// TIA Portal V18 program export: 1 tag tables, 1 data types, 3 data blocks, 17 code blocks (in call order from the OBs), 10 instance data blocks

VAR_GLOBAL   // PLC tag table "默认变量表"
   Room1_ES1 AT %I200.0 : Bool;
   Room1_ES2 AT %I200.1 : Bool;
   Room1_ES3 AT %I200.2 : Bool;
   Room1_ES4 AT %I200.3 : Bool;
   Room1_ES5 AT %I206.0 : Bool;
   Room1Control_ES6 AT %I206.1 : Bool;
   "Room1_Key1.1" AT %I206.2 : Bool;
   "Room1Control_Key1.1" AT %I206.3 : Bool;
   "Room1_door1.1" AT %I212.0 : Bool;
   Room2_ES1 AT %I218.0 : Bool;
   Room2_ES2 AT %I218.1 : Bool;
   Room2_ES3 AT %I218.2 : Bool;
   Room2_ES4 AT %I218.3 : Bool;
   Room2_ES5 AT %I224.0 : Bool;
   Room2Control_ES6 AT %I224.1 : Bool;
   "Room2_Key1.1" AT %I224.2 : Bool;
   "Room2Control_Key1.1" AT %I224.3 : Bool;
   "Room2_door1.1" AT %I230.0 : Bool;
   ACC_ES1 AT %I236.0 : Bool;
   ACC_ES2 AT %I236.1 : Bool;
   ACC_ES3 AT %I236.2 : Bool;
   ACC_ES4 AT %I236.3 : Bool;
   "ACC_Key1.1" AT %I242.2 : Bool;
   "ACCControl_Key1.1" AT %I242.3 : Bool;
   "ACC_door1.1" AT %I248.0 : Bool;
   "ACC_door2.1" AT %I248.1 : Bool;
   VerticalBeam_ES1 AT %I254.0 : Bool;   // vertical beam ES
   VerticalBeam_ES2 AT %I254.1 : Bool;
   VerticalBeam_ES3 AT %I254.2 : Bool;
   VerticalBeam_ES4 AT %I254.3 : Bool;
   "VerticalBeam_Key1.1" AT %I260.2 : Bool;
   "VerticalBeamControl_Key1.1" AT %I260.3 : Bool;
   "VerticalBeam_door1.1" AT %I266.0 : Bool;
   "VerticalBeam_door2.1" AT %I266.1 : Bool;
   Room1_SB1 AT %I100.0 : Bool;   // 搜索清场按钮1
   Room1_SB2 AT %I100.1 : Bool;
   Room2_SB1 AT %I100.4 : Bool;
   Room2_SB2 AT %I100.5 : Bool;
   ACC_SB1 AT %I101.0 : Bool;
   ACC_SB2 AT %I101.1 : Bool;
   VerticalBeam_SB1 AT %I101.4 : Bool;
   VerticalBeam_SB2 AT %I101.5 : Bool;
   ACC_Ready AT %I102.0 : Bool;
   ACC_Run AT %I102.1 : Bool;
   ACC_StopBeam AT %I102.2 : Bool;
   ACC_Stop AT %I102.3 : Bool;
   ACC_Fault AT %I102.4 : Bool;
   ACC_Mode1 AT %I102.5 : Bool;   // 治疗室1、加速器2、垂直束
   ACC_Mode2 AT %I102.6 : Bool;   // 治疗室2、加速器2、垂直束
   ACC_Mode3 AT %I102.7 : Bool;   // 加速器2、垂直束
   EnvironmentalMonitoring1 AT %I103.4 : Bool;
   EnvironmentalMonitoring2 AT %I103.5 : Bool;
   EnvironmentalMonitoring3 AT %I103.6 : Bool;
   EnvironmentalMonitoring4 AT %I103.7 : Bool;
   Room1_AudibleAlarm AT %Q100.0 : Bool;
   Room1_StrobeLamp1 AT %Q100.1 : Bool;
   Room1_StrobeLamp2 AT %Q100.2 : Bool;
   Room1_Red AT %Q100.5 : Bool;   // 禁止进入指示灯
   Room1_Yellow AT %Q100.6 : Bool;   // 限制进入指示灯
   Room1_Green AT %Q100.7 : Bool;   // 控制进入指示灯
   Room1_Door1NoEntry AT %Q101.0 : Bool;   // 门禁1禁止进入
   Room1_Door1RestrictedEntry AT %Q101.1 : Bool;   // 门禁1限制进入
   Room1_Door1ControlEntry AT %Q101.2 : Bool;   // 门禁1控制进入
   "Room1_door1.2" AT %I212.4 : Bool;
   "Room1_Key1.2" AT %I206.6 : Bool;
   "Room1Control_Key1.2" AT %I206.7 : Bool;
   "Room2_Key1.2" AT %I224.6 : Bool;
   "Room2Control_Key1.2" AT %I224.7 : Bool;
   "Room2_door1.2" AT %I230.4 : Bool;
   "ACC_Key1.2" AT %I242.6 : Bool;
   "ACCControl_Key1.2" AT %I242.7 : Bool;
   "VerticalBeam_Key1.2" AT %I260.6 : Bool;
   "VerticalBeamControl_Key1.2" AT %I260.7 : Bool;
   "VerticalBeam_door1.2" AT %I266.4 : Bool;
   "VerticalBeam_door2.2" AT %I266.5 : Bool;
   "ACC_door1.2" AT %I248.4 : Bool;
   "ACC_door2.2" AT %I248.5 : Bool;
   ACC_Interlock1 AT %Q400.0 : Bool;
   ACC_Interlock2 AT %Q400.1 : Bool;
   RF_Interlock1 AT %Q400.2 : Bool;
   RF_Interlock2 AT %Q400.3 : Bool;
   IonSource_Interlock1 AT %Q400.4 : Bool;
   IonSource_Interlock2 AT %Q400.5 : Bool;
   MIS__Interlock1 AT %Q400.6 : Bool;
   MIS__Interlock2 AT %Q400.7 : Bool;
   Room1_ES1_ValueStatus AT %I201.0 : Bool;
   Room1_ES2_ValueStatus AT %I201.1 : Bool;
   Room1_ES3_ValueStatus AT %I201.2 : Bool;
   Room1_ES4_ValueStatus AT %I201.3 : Bool;
   Room1_ES5_ValueStatus AT %I207.0 : Bool;
   Room1Control_ES6_ValueStatus AT %I207.1 : Bool;
   "Room1_Key1.1_ValueStatus" AT %I207.2 : Bool;
   "Room1Control_Key1.1_ValueStatus" AT %I207.3 : Bool;
   "Room1_Key1.2_ValueStatus" AT %I207.6 : Bool;
   "Room1Control_Key1.2_ValueStatus" AT %I207.7 : Bool;
   "Room1_door1.1_ValueStatus" AT %I213.0 : Bool;
   "Room1_door1.2_ValueStatus" AT %I213.4 : Bool;
   Room2_ES1_ValueStatus AT %I219.0 : Bool;
   Room2_ES2_ValueStatus AT %I219.1 : Bool;
   Room2_ES3_ValueStatus AT %I219.2 : Bool;
   Room2_ES4_ValueStatus AT %I219.3 : Bool;
   Room2_ES5_ValueStatus AT %I225.0 : Bool;
   Room2Control_ES6_ValueStatus AT %I225.1 : Bool;
   "Room2_Key1.1_ValueStatus" AT %I225.2 : Bool;
   "Room2Control_Key1.1_ValueStatus" AT %I225.3 : Bool;
   "Room2_Key1.2_ValueStatus" AT %I225.6 : Bool;
   "Room2Control_Key1.2_ValueStatus" AT %I225.7 : Bool;
   "Room2_door1.1_ValueStatus" AT %I231.0 : Bool;
   "Room2_door1.2_ValueStatus" AT %I231.4 : Bool;
   ACC_ES1_ValueStatus AT %I237.0 : Bool;
   ACC_ES2_ValueStatus AT %I237.1 : Bool;
   ACC_ES3_ValueStatus AT %I237.2 : Bool;
   ACC_ES4_ValueStatus AT %I237.3 : Bool;
   "ACC_Key1.1_ValueStatus" AT %I243.2 : Bool;
   "ACCControl_Key1.1_ValueStatus" AT %I243.3 : Bool;
   "ACC_Key1.2_ValueStatus" AT %I243.6 : Bool;
   "ACCControl_Key1.2_ValueStatus" AT %I243.7 : Bool;
   "ACC_door1.1_ValueStatus" AT %I249.0 : Bool;
   "ACC_door2.1_ValueStatus" AT %I249.1 : Bool;
   "ACC_door1.2_ValueStatus" AT %I249.4 : Bool;
   "ACC_door2.2_ValueStatus" AT %I249.5 : Bool;
   VerticalBeam_ES1_ValueStatus AT %I255.0 : Bool;
   VerticalBeam_ES2_ValueStatus AT %I255.1 : Bool;
   VerticalBeam_ES3_ValueStatus AT %I255.2 : Bool;
   VerticalBeam_ES4_ValueStatus AT %I255.3 : Bool;
   "VerticalBeam_Key1.1_ValueStatus" AT %I261.2 : Bool;
   "VerticalBeamControl_Key1.1_ValueStatus" AT %I261.3 : Bool;
   "VerticalBeam_Key1.2_ValueStatus" AT %I261.6 : Bool;
   "VerticalBeamControl_Key1.2_ValueStatus" AT %I261.7 : Bool;
   "VerticalBeam_door1.1_ValueStatus" AT %I267.0 : Bool;
   "VerticalBeam_door2.1_ValueStatus" AT %I267.1 : Bool;
   "VerticalBeam_door1.2_ValueStatus" AT %I267.4 : Bool;
   "VerticalBeam_door2.2_ValueStatus" AT %I267.5 : Bool;
   ACC_Interlock1_ValueStatus AT %I400.0 : Bool;
   ACC_Interlock2_ValueStatus AT %I400.1 : Bool;
   RF_Interlock1_ValueStatus AT %I400.2 : Bool;
   RF_Interlock2_ValueStatus AT %I400.3 : Bool;
   IonSource_Interlock1_ValueStatus AT %I400.4 : Bool;
   IonSource_Interlock2_ValueStatus AT %I400.5 : Bool;
   MIS__Interlock1_ValueStatus AT %I400.6 : Bool;
   MIS__Interlock2_ValueStatus AT %I400.7 : Bool;
   Room2_AudibleAlarm AT %Q102.0 : Bool;
   Room2_StrobeLamp1 AT %Q102.1 : Bool;
   Room2_StrobeLamp2 AT %Q102.2 : Bool;
   Room2_Red AT %Q102.5 : Bool;
   Room2_Yellow AT %Q102.6 : Bool;
   Room2_Green AT %Q102.7 : Bool;
   Room2_Door1NoEntry AT %Q103.0 : Bool;
   Room2_Door1RestrictedEntry AT %Q103.1 : Bool;
   Room2_Door1ControlEntry AT %Q103.2 : Bool;
   ACC_AudibleAlarm AT %Q104.0 : Bool;
   ACC_StrobeLamp1 AT %Q104.1 : Bool;
   ACC_StrobeLamp2 AT %Q104.2 : Bool;
   ACC_Red AT %Q104.5 : Bool;
   ACC_Yellow AT %Q104.6 : Bool;
   ACC_Green AT %Q104.7 : Bool;
   ACC_StrobeLamp3 AT %Q104.3 : Bool;
   ACC_StrobeLamp4 AT %Q104.4 : Bool;
   ACC_Door1NoEntry AT %Q105.0 : Bool;
   ACC_Door1RestrictedEntry AT %Q105.1 : Bool;
   ACC_Door1ControlEntry AT %Q105.2 : Bool;
   ACC_Door2NoEntry AT %Q105.3 : Bool;
   ACC_Door2RestrictedEntry AT %Q105.4 : Bool;
   ACC_Door2ControlEntry AT %Q105.5 : Bool;
   VerticalBeam_AudibleAlarm AT %Q106.0 : Bool;
   VerticalBeam_StrobeLamp1 AT %Q106.1 : Bool;
   VerticalBeam_StrobeLamp2 AT %Q106.2 : Bool;
   VerticalBeam_StrobeLamp3 AT %Q106.3 : Bool;
   VerticalBeam_StrobeLamp4 AT %Q106.4 : Bool;
   VerticalBeam_Red AT %Q106.5 : Bool;
   VerticalBeam_Yellow AT %Q106.6 : Bool;
   VerticalBeam_Green AT %Q106.7 : Bool;
   VerticalBeam_Door1NoEntry AT %Q107.0 : Bool;
   VerticalBeam_Door1RestrictedEntry AT %Q107.1 : Bool;
   VerticalBeam_Door1ControlEntry AT %Q107.2 : Bool;
   VerticalBeam_Door2NoEntry AT %Q107.3 : Bool;
   VerticalBeam_Door2RestrictedEntry AT %Q107.4 : Bool;
   VerticalBeam_Door2ControlEntry AT %Q107.5 : Bool;
   Room1_AreaReady AT %Q108.0 : Bool;   // 治疗室1控制区就绪
   Room2_AreaReady AT %Q108.1 : Bool;   // 治疗室2控制区就绪
   ACC_AreaReady AT %Q108.2 : Bool;   // 加速器2控制区就绪
   Room1_StartAlarm AT %Q101.7 : Bool;
   Room2_StartAlarm AT %Q103.7 : Bool;
   ACC_StartAlarm AT %Q105.7 : Bool;
   VerticalBeam_StartAlarm AT %Q107.7 : Bool;
   Room1_BeamAllowed AT %Q108.4 : Bool;   // 允许治疗室1打靶
   Room2_BeamAllowed AT %Q108.5 : Bool;   // 允许治疗室2打靶
   ACC_BeamAllowed AT %Q108.6 : Bool;   // 允许加速器出束
   VerticalBeam_AreaReady AT %Q108.3 : Bool;   // 垂直束控制区就绪
END_VAR

TYPE "FIODia"
// stored: IsFailsafeCompliant true
   STRUCT
      ModulePassOut : Bool;   // 模块钝化
      ModuleACK_REQ : Bool;   // 模块需确认重新集成
      Channel0PassOut : Bool;   // 通道0钝化
      Channel1PassOut : Bool;   // 通道1钝化
      Channel2PassOut : Bool;   // 通道2钝化
      Channel3PassOut : Bool;   // 通道3钝化
      Channel4PassOut : Bool;   // 通道4钝化
      Channel5PassOut : Bool;   // 通道5钝化
      Channel6PassOut : Bool;   // 通道6钝化
      Channel7PassOut : Bool;   // 通道7钝化
   END_STRUCT;
END_TYPE

DATA_BLOCK "数据块_1"   // DB2
{ S7_Optimized_Access := 'TRUE' }
VERSION : 0.1
// stored: AutoNumber true, DBAccessibleFromOPCUA true, IsOnlyStoredInLoadMemory false, IsRetainMemResEnabled false, IsWriteProtectedInAS false, MemoryReserve 100
   VAR
      Room1_Interlock : Bool;
      Room2_Interlock : Bool;
      ACC_Interlock : Bool;
      VerticalBeam_Interlock : Bool;
      Interlock : Bool;
   END_VAR
BEGIN
END_DATA_BLOCK

DATA_BLOCK "数据块_2"   // DB3
{ S7_Optimized_Access := 'TRUE' }
VERSION : 0.1
// stored: AutoNumber true, DBAccessibleFromOPCUA true, IsOnlyStoredInLoadMemory false, IsRetainMemResEnabled false, IsWriteProtectedInAS false, MemoryReserve 100
   VAR
      "F-DI_A21_1" : "FIODia";   // 安全输入模块A21.1
      "F-DI_A21_2" { S7_SetPoint := 'True'} : "FIODia";   // 安全输入模块A21.2
      "F-DI_A21_3" { S7_SetPoint := 'True'} : "FIODia";   // 安全输入模块A21.3
      "F-DI_A21_4" { S7_SetPoint := 'True'} : "FIODia";   // 安全输入模块A21.4
      "F-DI_A21_5" { S7_SetPoint := 'True'} : "FIODia";   // 安全输入模块A21.5
      "F-DI_A21_6" { S7_SetPoint := 'True'} : "FIODia";   // 安全输入模块A21.6
      "F-DI_A21_7" { S7_SetPoint := 'True'} : "FIODia";   // 安全输入模块A21.7
      "F-DI_A21_8" { S7_SetPoint := 'True'} : "FIODia";   // 安全输入模块A21.8
      "F-DI_A21_9" { S7_SetPoint := 'True'} : "FIODia";   // 安全输入模块A21.9
      "F-DI_A21_10" { S7_SetPoint := 'True'} : "FIODia";   // 安全输入模块A21.10
      "F-DI_A21_11" { S7_SetPoint := 'True'} : "FIODia";   // 安全输入模块A21.11
      "F-DI_A21_12" { S7_SetPoint := 'True'} : "FIODia";   // 安全输入模块A21.12
      "F-DQ_A21_1" { S7_SetPoint := 'True'} : "FIODia";   // 安全输出模块A22.1
      "F-DQ_A21_2" { S7_SetPoint := 'True'} : "FIODia";   // 安全输出模块A22.2
   END_VAR
BEGIN
END_DATA_BLOCK

DATA_BLOCK "EPICSData"   // DB8
{ S7_Optimized_Access := 'FALSE'; DB_Accessible_From_OPC_UA := 'FALSE' }
VERSION : 0.1
// stored: AutoNumber true, DBAccessibleFromOPCUA false, IsOnlyStoredInLoadMemory false, IsWriteProtectedInAS false
   VAR
      Reset : Bool;
   END_VAR
BEGIN
END_DATA_BLOCK

ORGANIZATION_BLOCK "Main"   // OB1, LAD, ProgramCycle
TITLE = "Main Program Sweep (Cycle)"
{ S7_Optimized_Access := 'TRUE' }
VERSION : 0.1
// stored: AutoNumber true, IsIECCheckEnabled false, SetENOAutomatically false
   VAR_INPUT
      Initial_Call : Bool;   // Initial call of this OB
      Remanence : Bool;   // =True, if remanent data are available
   END_VAR
BEGIN

REGION Network 2
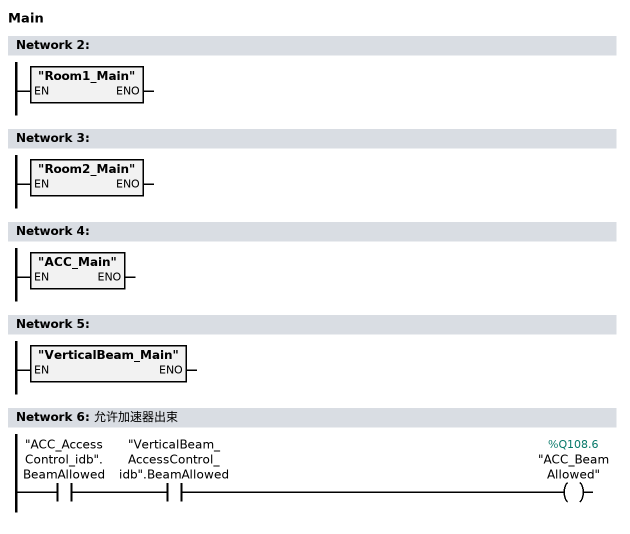
   RUNG wire#powerrail
      "Room1_Main"()
   END_RUNG
   // the same network as SCL:
   "Room1_Main"();
END_REGION

REGION Network 3
   RUNG wire#powerrail
      "Room2_Main"()
   END_RUNG
   // the same network as SCL:
   "Room2_Main"();
END_REGION

REGION Network 4
   RUNG wire#powerrail
      "ACC_Main"()
   END_RUNG
   // the same network as SCL:
   "ACC_Main"();
END_REGION

REGION Network 5
   RUNG wire#powerrail
      "VerticalBeam_Main"()
   END_RUNG
   // the same network as SCL:
   "VerticalBeam_Main"();
END_REGION

REGION Network 6: 允许加速器出束
   RUNG wire#powerrail
      Contact( "ACC_AccessControl_idb".BeamAllowed )
      Contact( "VerticalBeam_AccessControl_idb".BeamAllowed )
      Coil( "ACC_BeamAllowed" )
   END_RUNG
   // the same network as SCL:
   "ACC_BeamAllowed" := "ACC_AccessControl_idb".BeamAllowed AND "VerticalBeam_AccessControl_idb".BeamAllowed;
END_REGION
END_ORGANIZATION_BLOCK

FUNCTION "Room1_Main" : Void   // FC4, LAD
{ S7_Optimized_Access := 'TRUE' }
VERSION : 0.1
// stored: AutoNumber true, IsIECCheckEnabled false, SetENOAutomatically false, UDAEnableTagReadback false
BEGIN

REGION Network 1: 区域搜索
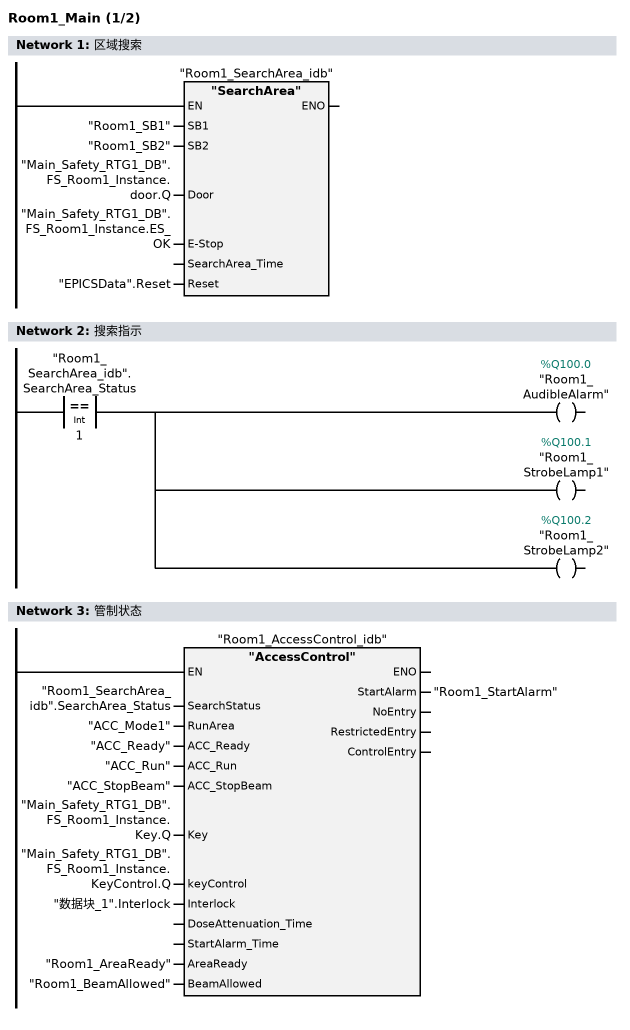
   RUNG wire#powerrail
      "Room1_SearchArea_idb"(SB1 := "Room1_SB1", SB2 := "Room1_SB2", Door := "Main_Safety_RTG1_DB".FS_Room1_Instance.door.Q, "E-Stop" := "Main_Safety_RTG1_DB".FS_Room1_Instance.ES_OK, SearchArea_Time :=, Reset := "EPICSData".Reset)
   END_RUNG
   // the same network as SCL:
   "Room1_SearchArea_idb"(SB1 := "Room1_SB1",   // "SearchArea"
                          SB2 := "Room1_SB2",
                          Door := "Main_Safety_RTG1_DB".FS_Room1_Instance.door.Q,
                          "E-Stop" := "Main_Safety_RTG1_DB".FS_Room1_Instance.ES_OK,
                          Reset := "EPICSData".Reset);
END_REGION

REGION Network 2: 搜索指示
   RUNG wire#powerrail
      { S7_Templates := "SrcType := Int" } EQ_Contact(in1 := "Room1_SearchArea_idb".SearchArea_Status, in2 := 1)
      wire#w1
      Coil( "Room1_AudibleAlarm" )
   END_RUNG
   RUNG wire#w1
      Coil( "Room1_StrobeLamp1" )
   END_RUNG
   RUNG wire#w1
      Coil( "Room1_StrobeLamp2" )
   END_RUNG
   // the same network as SCL:
   "Room1_AudibleAlarm" := "Room1_SearchArea_idb".SearchArea_Status = 1;
   "Room1_StrobeLamp1" := "Room1_AudibleAlarm";
   "Room1_StrobeLamp2" := "Room1_AudibleAlarm";
END_REGION

REGION Network 3: 管制状态
   RUNG wire#powerrail
      "Room1_AccessControl_idb"(SearchStatus := "Room1_SearchArea_idb".SearchArea_Status, RunArea := "ACC_Mode1", ACC_Ready := "ACC_Ready", ACC_Run := "ACC_Run", ACC_StopBeam := "ACC_StopBeam", Key := "Main_Safety_RTG1_DB".FS_Room1_Instance.Key.Q, keyControl := "Main_Safety_RTG1_DB".FS_Room1_Instance.KeyControl.Q, Interlock := "数据块_1".Interlock, DoseAttenuation_Time :=, StartAlarm_Time :=, AreaReady := "Room1_AreaReady", BeamAllowed := "Room1_BeamAllowed", StartAlarm => "Room1_StartAlarm", NoEntry =>, RestrictedEntry =>, ControlEntry =>)
   END_RUNG
   // the same network as SCL:
   "Room1_AccessControl_idb"(SearchStatus := "Room1_SearchArea_idb".SearchArea_Status,   // "AccessControl"
                           RunArea := "ACC_Mode1",
                           ACC_Ready := "ACC_Ready",
                           ACC_Run := "ACC_Run",
                           ACC_StopBeam := "ACC_StopBeam",
                           Key := "Main_Safety_RTG1_DB".FS_Room1_Instance.Key.Q,
                           keyControl := "Main_Safety_RTG1_DB".FS_Room1_Instance.KeyControl.Q,
                           Interlock := "数据块_1".Interlock,
                           AreaReady := "Room1_AreaReady",
                           BeamAllowed := "Room1_BeamAllowed",
                           StartAlarm => "Room1_StartAlarm");
END_REGION

REGION Network 4: 管制输出
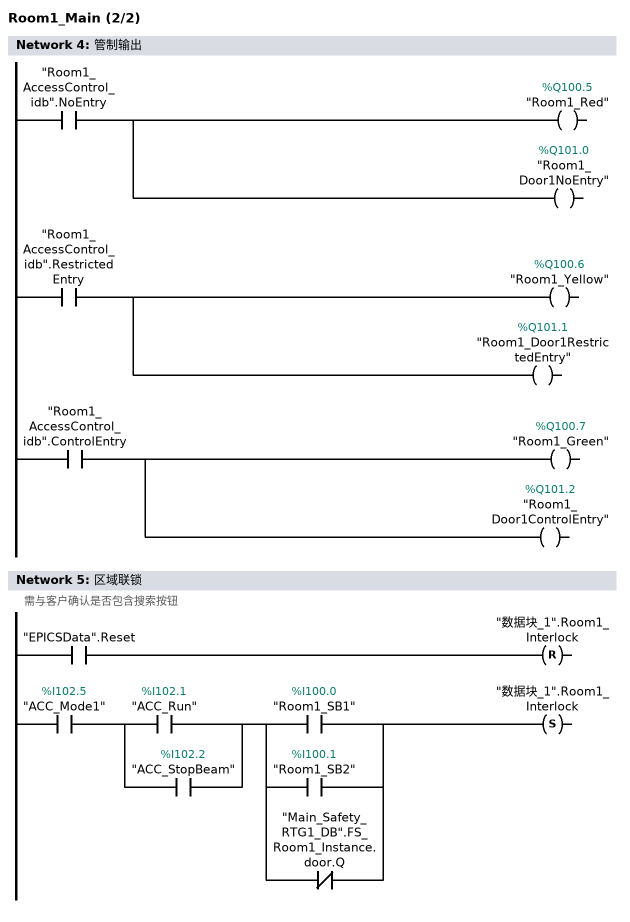
   RUNG wire#powerrail
      Contact( "Room1_AccessControl_idb".NoEntry )
      wire#w1
      Coil( "Room1_Red" )
   END_RUNG
   RUNG wire#w1
      Coil( "Room1_Door1NoEntry" )
   END_RUNG
   RUNG wire#powerrail
      Contact( "Room1_AccessControl_idb".RestrictedEntry )
      wire#w2
      Coil( "Room1_Yellow" )
   END_RUNG
   RUNG wire#w2
      Coil( "Room1_Door1RestrictedEntry" )
   END_RUNG
   RUNG wire#powerrail
      Contact( "Room1_AccessControl_idb".ControlEntry )
      wire#w3
      Coil( "Room1_Green" )
   END_RUNG
   RUNG wire#w3
      Coil( "Room1_Door1ControlEntry" )
   END_RUNG
   // the same network as SCL:
   "Room1_Red" := "Room1_AccessControl_idb".NoEntry;
   "Room1_Door1NoEntry" := "Room1_AccessControl_idb".NoEntry;
   "Room1_Yellow" := "Room1_AccessControl_idb".RestrictedEntry;
   "Room1_Door1RestrictedEntry" := "Room1_AccessControl_idb".RestrictedEntry;
   "Room1_Green" := "Room1_AccessControl_idb".ControlEntry;
   "Room1_Door1ControlEntry" := "Room1_AccessControl_idb".ControlEntry;
END_REGION

REGION Network 5: 区域联锁
   // 需与客户确认是否包含搜索按钮
   RUNG wire#powerrail
      Contact( "EPICSData".Reset )
      R_Coil( "数据块_1".Room1_Interlock )
   END_RUNG
   RUNG wire#powerrail
      Contact( "ACC_Mode1" )
      wire#w1
      Contact( "ACC_Run" )
      wire#w2
      Contact( "Room1_SB1" )
      wire#w3
      S_Coil( "数据块_1".Room1_Interlock )
   END_RUNG
   RUNG wire#w1
      Contact( "ACC_StopBeam" )
   END_RUNG wire#w2
   RUNG wire#w2
      Contact( "Room1_SB2" )
   END_RUNG wire#w3
   RUNG wire#w2
      I_Contact( "Main_Safety_RTG1_DB".FS_Room1_Instance.door.Q )
   END_RUNG wire#w3
   // the same network as SCL:
   IF "EPICSData".Reset THEN "数据块_1".Room1_Interlock := FALSE; END_IF;
   IF "ACC_Mode1" AND ("ACC_Run" OR "ACC_StopBeam") AND ("Room1_SB1" OR "Room1_SB2" OR NOT "Main_Safety_RTG1_DB".FS_Room1_Instance.door.Q) THEN
       "数据块_1".Room1_Interlock := TRUE;
   END_IF;
END_REGION
END_FUNCTION

FUNCTION_BLOCK "SearchArea"   // FB6, LAD
{ S7_Optimized_Access := 'TRUE' }
VERSION : 0.1
// stored: AutoNumber true, IsIECCheckEnabled false, IsRetainMemResEnabled false, MemoryReserve 100, SetENOAutomatically false, UDAEnableTagReadback false
   VAR_INPUT
      SB1 : Bool;
      SB2 : Bool;
      Door : Bool;
      "E-Stop" : Bool;
      SearchArea_Time : Time := T#5m;
      Reset : Bool;
   END_VAR
   VAR
      SearchArea_Timer { S7_SetPoint := 'True'} : TON_TIME;
      SearchArea_Status : Int;   // 0:未搜索;1:搜索中;2:搜索完成;
      "Step" { S7_SetPoint := 'True'} : Int;
      Error { ExternalAccessible := 'False'; ExternalVisible := 'False'; ExternalWritable := 'False'} : Struct
         All { ExternalAccessible := 'False'; ExternalVisible := 'False'; ExternalWritable := 'False'} : Bool;   // 搜索总故障
         StartFail { ExternalAccessible := 'False'; ExternalVisible := 'False'; ExternalWritable := 'False'} : Bool;   // 搜索启动失败，请确认未按下搜索按钮2或未关闭门
         WrongSequence1 { ExternalAccessible := 'False'; ExternalVisible := 'False'; ExternalWritable := 'False'} : Bool;   // 搜索顺序错误，此时应按下搜索按钮2，请勿按搜索按钮1或关闭门
         WrongSequence2 { ExternalAccessible := 'False'; ExternalVisible := 'False'; ExternalWritable := 'False'} : Bool;   // 搜索顺序错误，此时应关闭门，请勿按搜索按钮1或搜索按钮2
         Timeout { ExternalAccessible := 'False'; ExternalVisible := 'False'; ExternalWritable := 'False'} : Bool;   // 搜索超时
      END_STRUCT;
   END_VAR
   VAR_TEMP   // added for the SCL form of the ladder/FBD networks
      _w1 : Bool;
   END_VAR
BEGIN

REGION Network 1: 搜索破坏
   // 搜索完成后，当搜索按钮按下，门被打开，急停按钮按下，搜索状态设置为未搜索
   // 需与客户确认破坏条件是否包含搜索按钮和急停？
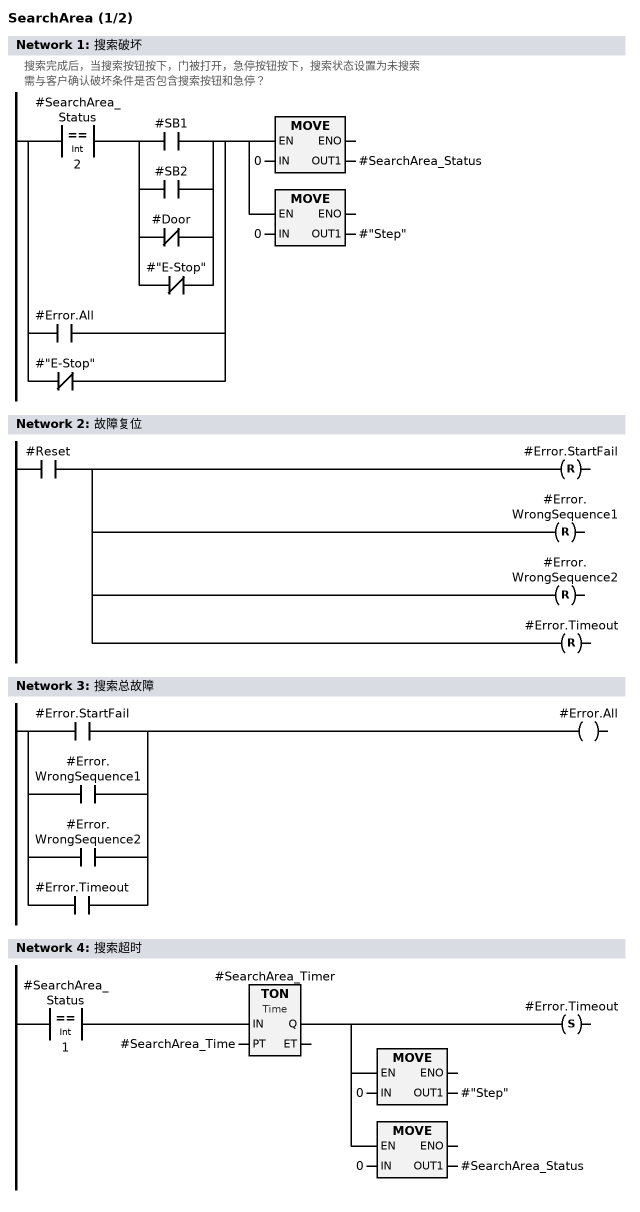
   RUNG wire#powerrail
      { S7_Templates := "SrcType := Int" } EQ_Contact(in1 := #SearchArea_Status, in2 := 2)
      wire#w1
      Contact( #SB1 )
      wire#w2
      Move(in := 0, out1 => #SearchArea_Status)
   END_RUNG
   RUNG wire#w1
      Contact( #SB2 )
   END_RUNG wire#w2
   RUNG wire#w1
      I_Contact( #Door )
   END_RUNG wire#w2
   RUNG wire#w1
      I_Contact( #"E-Stop" )
   END_RUNG wire#w2
   RUNG wire#powerrail
      Contact( #Error.All )
   END_RUNG wire#w2
   RUNG wire#powerrail
      I_Contact( #"E-Stop" )
   END_RUNG wire#w2
   RUNG wire#w2
      Move(in := 0, out1 => #"Step")
   END_RUNG
   // the same network as SCL:
   #_w1 := ((#SearchArea_Status = 2) AND (#SB1 OR #SB2 OR NOT #Door OR NOT #"E-Stop")) OR #Error.All OR NOT #"E-Stop";
   IF #_w1 THEN
       #SearchArea_Status := 0;
       #"Step" := 0;
   END_IF;
END_REGION

REGION Network 2: 故障复位
   RUNG wire#powerrail
      Contact( #Reset )
      wire#w1
      R_Coil( #Error.StartFail )
   END_RUNG
   RUNG wire#w1
      R_Coil( #Error.WrongSequence1 )
   END_RUNG
   RUNG wire#w1
      R_Coil( #Error.WrongSequence2 )
   END_RUNG
   RUNG wire#w1
      R_Coil( #Error.Timeout )
   END_RUNG
   // the same network as SCL:
   IF #Reset THEN
       #Error.StartFail := FALSE;
       #Error.WrongSequence1 := FALSE;
       #Error.WrongSequence2 := FALSE;
       #Error.Timeout := FALSE;
   END_IF;
END_REGION

REGION Network 3: 搜索总故障
   RUNG wire#powerrail
      Contact( #Error.StartFail )
      wire#w1
      Coil( #Error.All )
   END_RUNG
   RUNG wire#powerrail
      Contact( #Error.WrongSequence1 )
   END_RUNG wire#w1
   RUNG wire#powerrail
      Contact( #Error.WrongSequence2 )
   END_RUNG wire#w1
   RUNG wire#powerrail
      Contact( #Error.Timeout )
   END_RUNG wire#w1
   // the same network as SCL:
   #Error.All := #Error.StartFail OR #Error.WrongSequence1 OR #Error.WrongSequence2 OR #Error.Timeout;
END_REGION

REGION Network 4: 搜索超时
   RUNG wire#powerrail
      { S7_Templates := "SrcType := Int" } EQ_Contact(in1 := #SearchArea_Status, in2 := 1)
      { S7_Templates := "time_type := Time" } #SearchArea_Timer.TON(pt := #SearchArea_Time, et =>)
      wire#w1
      S_Coil( #Error.Timeout )
   END_RUNG
   RUNG wire#w1
      Move(in := 0, out1 => #"Step")
   END_RUNG
   RUNG wire#w1
      Move(in := 0, out1 => #SearchArea_Status)
   END_RUNG
   // the same network as SCL:
   #SearchArea_Timer(IN := #SearchArea_Status = 1, PT := #SearchArea_Time);   // TON
   IF #SearchArea_Timer.Q THEN
       #Error.Timeout := TRUE;
       #"Step" := 0;
       #SearchArea_Status := 0;
   END_IF;
END_REGION

REGION Network 5: 按下SB1，开始搜索
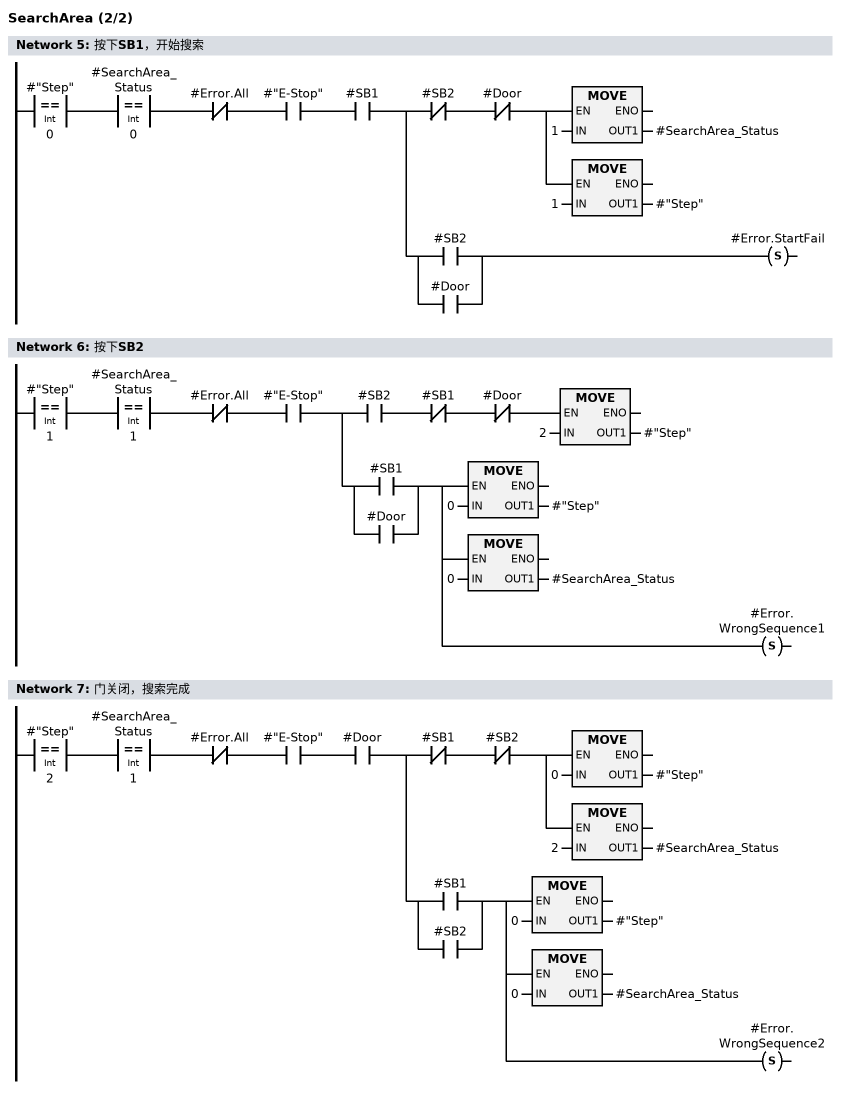
   RUNG wire#powerrail
      { S7_Templates := "SrcType := Int" } EQ_Contact(in1 := #"Step", in2 := 0)
      { S7_Templates := "SrcType := Int" } EQ_Contact(in1 := #SearchArea_Status, in2 := 0)
      I_Contact( #Error.All )
      Contact( #"E-Stop" )
      Contact( #SB1 )
      wire#w1
      I_Contact( #SB2 )
      I_Contact( #Door )
      wire#w2
      Move(in := 1, out1 => #SearchArea_Status)
   END_RUNG
   RUNG wire#w2
      Move(in := 1, out1 => #"Step")
   END_RUNG
   RUNG wire#w1
      Contact( #SB2 )
      wire#w3
      S_Coil( #Error.StartFail )
   END_RUNG
   RUNG wire#w1
      Contact( #Door )
   END_RUNG wire#w3
   // the same network as SCL:
   #_w1 := (#"Step" = 0) AND (#SearchArea_Status = 0) AND NOT #Error.All AND #"E-Stop" AND #SB1;
   IF #_w1 AND NOT #SB2 AND NOT #Door THEN
       #SearchArea_Status := 1;
       #"Step" := 1;
   END_IF;
   IF #_w1 AND (#SB2 OR #Door) THEN #Error.StartFail := TRUE; END_IF;
END_REGION

REGION Network 6: 按下SB2
   RUNG wire#powerrail
      { S7_Templates := "SrcType := Int" } EQ_Contact(in1 := #"Step", in2 := 1)
      { S7_Templates := "SrcType := Int" } EQ_Contact(in1 := #SearchArea_Status, in2 := 1)
      I_Contact( #Error.All )
      Contact( #"E-Stop" )
      wire#w1
      Contact( #SB2 )
      I_Contact( #SB1 )
      I_Contact( #Door )
      Move(in := 2, out1 => #"Step")
   END_RUNG
   RUNG wire#w1
      Contact( #SB1 )
      wire#w2
      Move(in := 0, out1 => #"Step")
   END_RUNG
   RUNG wire#w1
      Contact( #Door )
   END_RUNG wire#w2
   RUNG wire#w2
      Move(in := 0, out1 => #SearchArea_Status)
   END_RUNG
   RUNG wire#w2
      S_Coil( #Error.WrongSequence1 )
   END_RUNG
   // the same network as SCL:
   #_w1 := (#"Step" = 1) AND (#SearchArea_Status = 1) AND NOT #Error.All AND #"E-Stop";
   IF #_w1 AND #SB2 AND NOT #SB1 AND NOT #Door THEN #"Step" := 2; END_IF;
   IF #_w1 AND (#SB1 OR #Door) THEN
       #"Step" := 0;
       #SearchArea_Status := 0;
       #Error.WrongSequence1 := TRUE;
   END_IF;
END_REGION

REGION Network 7: 门关闭，搜索完成
   RUNG wire#powerrail
      { S7_Templates := "SrcType := Int" } EQ_Contact(in1 := #"Step", in2 := 2)
      { S7_Templates := "SrcType := Int" } EQ_Contact(in1 := #SearchArea_Status, in2 := 1)
      I_Contact( #Error.All )
      Contact( #"E-Stop" )
      Contact( #Door )
      wire#w1
      I_Contact( #SB1 )
      I_Contact( #SB2 )
      wire#w2
      Move(in := 0, out1 => #"Step")
   END_RUNG
   RUNG wire#w2
      Move(in := 2, out1 => #SearchArea_Status)
   END_RUNG
   RUNG wire#w1
      Contact( #SB1 )
      wire#w3
      Move(in := 0, out1 => #"Step")
   END_RUNG
   RUNG wire#w1
      Contact( #SB2 )
   END_RUNG wire#w3
   RUNG wire#w3
      Move(in := 0, out1 => #SearchArea_Status)
   END_RUNG
   RUNG wire#w3
      S_Coil( #Error.WrongSequence2 )
   END_RUNG
   // the same network as SCL:
   #_w1 := (#"Step" = 2) AND (#SearchArea_Status = 1) AND NOT #Error.All AND #"E-Stop" AND #Door;
   IF #_w1 AND NOT #SB1 AND NOT #SB2 THEN
       #"Step" := 0;
       #SearchArea_Status := 2;
   END_IF;
   IF #_w1 AND (#SB1 OR #SB2) THEN
       #"Step" := 0;
       #SearchArea_Status := 0;
       #Error.WrongSequence2 := TRUE;
   END_IF;
END_REGION
END_FUNCTION_BLOCK

FUNCTION_BLOCK "AccessControl"   // FB7, LAD
{ S7_Optimized_Access := 'TRUE' }
VERSION : 0.1
// stored: AutoNumber true, IsIECCheckEnabled false, IsRetainMemResEnabled false, MemoryReserve 100, SetENOAutomatically false, UDAEnableTagReadback false
   VAR_INPUT
      SearchStatus : Int;   // 0:未搜索;1:搜索中;2:搜索完成;
      RunArea : Bool;
      ACC_Ready : Bool;
      ACC_Run : Bool;
      ACC_StopBeam : Bool;
      Key : Bool;
      keyControl : Bool;
      Interlock : Bool;
      DoseAttenuation_Time : Time := T#1m;
      StartAlarm_Time : Time := T#2m;
   END_VAR
   VAR_OUTPUT
      StartAlarm : Bool;
      NoEntry : Bool;
      RestrictedEntry : Bool;
      ControlEntry : Bool;
   END_VAR
   VAR_IN_OUT
      AreaReady : Bool;
      BeamAllowed : Bool;
   END_VAR
   VAR
      State : Int;   // 0:禁止进入;1:限制进入;2:控制进入
      DoseAttenuation_Timer { S7_SetPoint := 'True'} : TON_TIME;
      StartAlarm_Timer { S7_SetPoint := 'True'} : TON_TIME;
   END_VAR
   VAR_TEMP   // added for the SCL form of the ladder/FBD networks
      _w1 : Bool;
   END_VAR
BEGIN

REGION Network 1
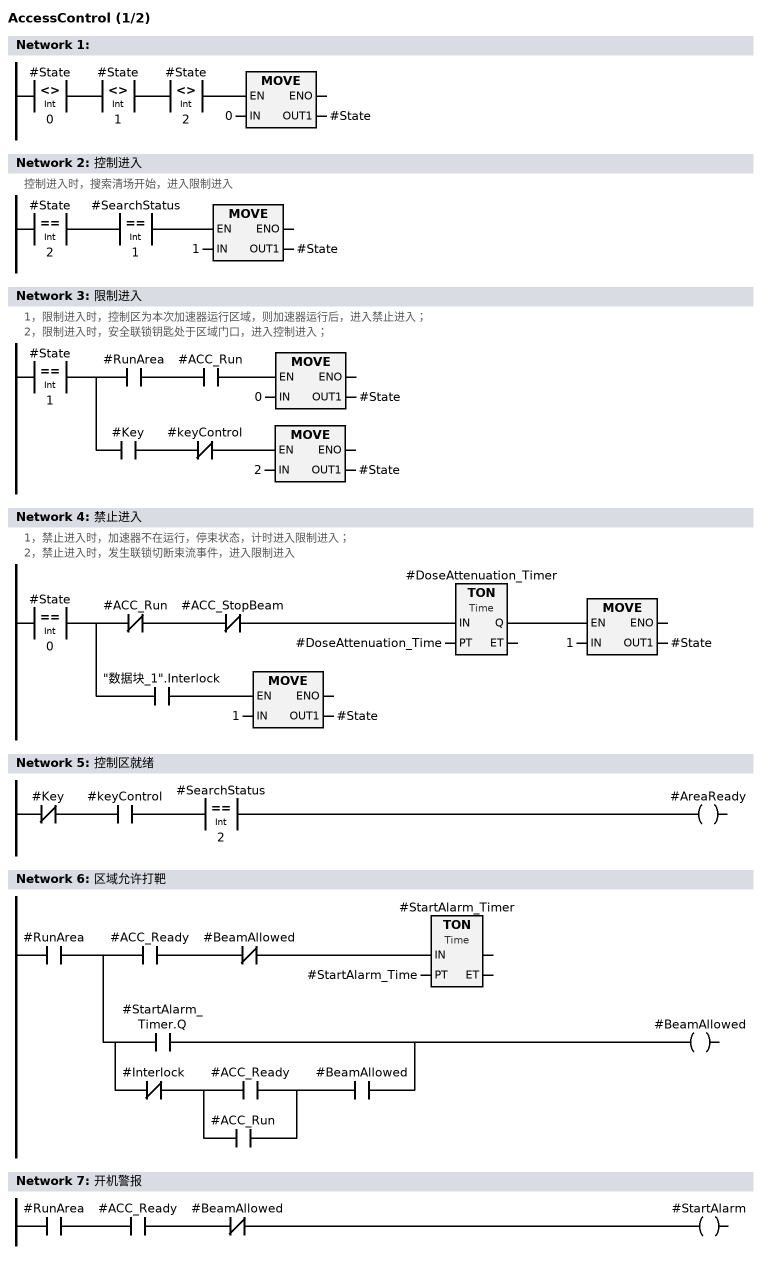
   RUNG wire#powerrail
      { S7_Templates := "SrcType := Int" } NE_Contact(in1 := #State, in2 := 0)
      { S7_Templates := "SrcType := Int" } NE_Contact(in1 := #State, in2 := 1)
      { S7_Templates := "SrcType := Int" } NE_Contact(in1 := #State, in2 := 2)
      Move(in := 0, out1 => #State)
   END_RUNG
   // the same network as SCL:
   IF (#State <> 0) AND (#State <> 1) AND (#State <> 2) THEN #State := 0; END_IF;
END_REGION

REGION Network 2: 控制进入
   // 控制进入时，搜索清场开始，进入限制进入
   RUNG wire#powerrail
      { S7_Templates := "SrcType := Int" } EQ_Contact(in1 := #State, in2 := 2)
      { S7_Templates := "SrcType := Int" } EQ_Contact(in1 := #SearchStatus, in2 := 1)
      Move(in := 1, out1 => #State)
   END_RUNG
   // the same network as SCL:
   IF (#State = 2) AND (#SearchStatus = 1) THEN #State := 1; END_IF;
END_REGION

REGION Network 3: 限制进入
   // 1，限制进入时，控制区为本次加速器运行区域，则加速器运行后，进入禁止进入；
   // 2，限制进入时，安全联锁钥匙处于区域门口，进入控制进入；
   RUNG wire#powerrail
      { S7_Templates := "SrcType := Int" } EQ_Contact(in1 := #State, in2 := 1)
      wire#w1
      Contact( #RunArea )
      Contact( #ACC_Run )
      Move(in := 0, out1 => #State)
   END_RUNG
   RUNG wire#w1
      Contact( #Key )
      I_Contact( #keyControl )
      Move(in := 2, out1 => #State)
   END_RUNG
   // the same network as SCL:
   #_w1 := #State = 1;
   IF #_w1 AND #RunArea AND #ACC_Run THEN #State := 0; END_IF;
   IF #_w1 AND #Key AND NOT #keyControl THEN #State := 2; END_IF;
END_REGION

REGION Network 4: 禁止进入
   // 1，禁止进入时，加速器不在运行，停束状态，计时进入限制进入；
   // 2，禁止进入时，发生联锁切断束流事件，进入限制进入
   RUNG wire#powerrail
      { S7_Templates := "SrcType := Int" } EQ_Contact(in1 := #State, in2 := 0)
      wire#w1
      I_Contact( #ACC_Run )
      I_Contact( #ACC_StopBeam )
      { S7_Templates := "time_type := Time" } #DoseAttenuation_Timer.TON(pt := #DoseAttenuation_Time, et =>)
      Move(in := 1, out1 => #State)
   END_RUNG
   RUNG wire#w1
      Contact( "数据块_1".Interlock )
      Move(in := 1, out1 => #State)
   END_RUNG
   // the same network as SCL:
   #_w1 := #State = 0;
   #DoseAttenuation_Timer(IN := #_w1 AND NOT #ACC_Run AND NOT #ACC_StopBeam, PT := #DoseAttenuation_Time);   // TON
   IF #DoseAttenuation_Timer.Q THEN #State := 1; END_IF;
   IF #_w1 AND "数据块_1".Interlock THEN #State := 1; END_IF;
END_REGION

REGION Network 5: 控制区就绪
   RUNG wire#powerrail
      I_Contact( #Key )
      Contact( #keyControl )
      { S7_Templates := "SrcType := Int" } EQ_Contact(in1 := #SearchStatus, in2 := 2)
      Coil( #AreaReady )
   END_RUNG
   // the same network as SCL:
   #AreaReady := NOT #Key AND #keyControl AND (#SearchStatus = 2);
END_REGION

REGION Network 6: 区域允许打靶
   RUNG wire#powerrail
      Contact( #RunArea )
      wire#w1
      Contact( #ACC_Ready )
      I_Contact( #BeamAllowed )
      { S7_Templates := "time_type := Time" } #StartAlarm_Timer.TON(pt := #StartAlarm_Time, et =>)
   END_RUNG
   RUNG wire#w1
      Contact( #StartAlarm_Timer.Q )
      wire#w2
      Coil( #BeamAllowed )
   END_RUNG
   RUNG wire#w1
      I_Contact( #Interlock )
      wire#w3
      Contact( #ACC_Ready )
      wire#w4
      Contact( #BeamAllowed )
   END_RUNG wire#w2
   RUNG wire#w3
      Contact( #ACC_Run )
   END_RUNG wire#w4
   // the same network as SCL:
   #StartAlarm_Timer(IN := #RunArea AND #ACC_Ready AND NOT #BeamAllowed, PT := #StartAlarm_Time);   // TON
   #BeamAllowed := #RunArea AND (#StartAlarm_Timer.Q OR (NOT #Interlock AND (#ACC_Ready OR #ACC_Run) AND #BeamAllowed));
END_REGION

REGION Network 7: 开机警报
   RUNG wire#powerrail
      Contact( #RunArea )
      Contact( #ACC_Ready )
      I_Contact( #BeamAllowed )
      Coil( #StartAlarm )
   END_RUNG
   // the same network as SCL:
   #StartAlarm := #RunArea AND #ACC_Ready AND NOT #BeamAllowed;
END_REGION

REGION Network 8
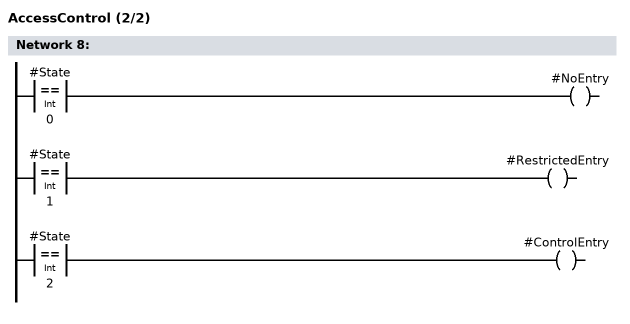
   RUNG wire#powerrail
      { S7_Templates := "SrcType := Int" } EQ_Contact(in1 := #State, in2 := 0)
      Coil( #NoEntry )
   END_RUNG
   RUNG wire#powerrail
      { S7_Templates := "SrcType := Int" } EQ_Contact(in1 := #State, in2 := 1)
      Coil( #RestrictedEntry )
   END_RUNG
   RUNG wire#powerrail
      { S7_Templates := "SrcType := Int" } EQ_Contact(in1 := #State, in2 := 2)
      Coil( #ControlEntry )
   END_RUNG
   // the same network as SCL:
   #NoEntry := #State = 0;
   #RestrictedEntry := #State = 1;
   #ControlEntry := #State = 2;
END_REGION
END_FUNCTION_BLOCK

FUNCTION "Room2_Main" : Void   // FC5, LAD
{ S7_Optimized_Access := 'TRUE' }
VERSION : 0.1
// stored: AutoNumber true, IsIECCheckEnabled false, SetENOAutomatically false, UDAEnableTagReadback false
BEGIN

REGION Network 1: 区域搜索
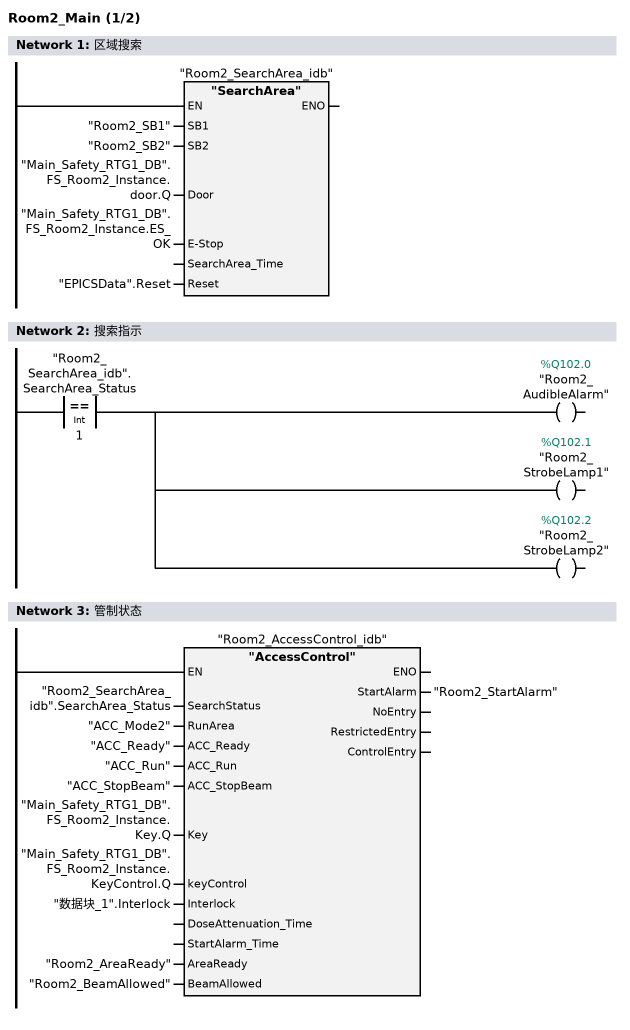
   RUNG wire#powerrail
      "Room2_SearchArea_idb"(SB1 := "Room2_SB1", SB2 := "Room2_SB2", Door := "Main_Safety_RTG1_DB".FS_Room2_Instance.door.Q, "E-Stop" := "Main_Safety_RTG1_DB".FS_Room2_Instance.ES_OK, SearchArea_Time :=, Reset := "EPICSData".Reset)
   END_RUNG
   // the same network as SCL:
   "Room2_SearchArea_idb"(SB1 := "Room2_SB1",   // "SearchArea"
                          SB2 := "Room2_SB2",
                          Door := "Main_Safety_RTG1_DB".FS_Room2_Instance.door.Q,
                          "E-Stop" := "Main_Safety_RTG1_DB".FS_Room2_Instance.ES_OK,
                          Reset := "EPICSData".Reset);
END_REGION

REGION Network 2: 搜索指示
   RUNG wire#powerrail
      { S7_Templates := "SrcType := Int" } EQ_Contact(in1 := "Room2_SearchArea_idb".SearchArea_Status, in2 := 1)
      wire#w1
      Coil( "Room2_AudibleAlarm" )
   END_RUNG
   RUNG wire#w1
      Coil( "Room2_StrobeLamp1" )
   END_RUNG
   RUNG wire#w1
      Coil( "Room2_StrobeLamp2" )
   END_RUNG
   // the same network as SCL:
   "Room2_AudibleAlarm" := "Room2_SearchArea_idb".SearchArea_Status = 1;
   "Room2_StrobeLamp1" := "Room2_AudibleAlarm";
   "Room2_StrobeLamp2" := "Room2_AudibleAlarm";
END_REGION

REGION Network 3: 管制状态
   RUNG wire#powerrail
      "Room2_AccessControl_idb"(SearchStatus := "Room2_SearchArea_idb".SearchArea_Status, RunArea := "ACC_Mode2", ACC_Ready := "ACC_Ready", ACC_Run := "ACC_Run", ACC_StopBeam := "ACC_StopBeam", Key := "Main_Safety_RTG1_DB".FS_Room2_Instance.Key.Q, keyControl := "Main_Safety_RTG1_DB".FS_Room2_Instance.KeyControl.Q, Interlock := "数据块_1".Interlock, DoseAttenuation_Time :=, StartAlarm_Time :=, AreaReady := "Room2_AreaReady", BeamAllowed := "Room2_BeamAllowed", StartAlarm => "Room2_StartAlarm", NoEntry =>, RestrictedEntry =>, ControlEntry =>)
   END_RUNG
   // the same network as SCL:
   "Room2_AccessControl_idb"(SearchStatus := "Room2_SearchArea_idb".SearchArea_Status,   // "AccessControl"
                           RunArea := "ACC_Mode2",
                           ACC_Ready := "ACC_Ready",
                           ACC_Run := "ACC_Run",
                           ACC_StopBeam := "ACC_StopBeam",
                           Key := "Main_Safety_RTG1_DB".FS_Room2_Instance.Key.Q,
                           keyControl := "Main_Safety_RTG1_DB".FS_Room2_Instance.KeyControl.Q,
                           Interlock := "数据块_1".Interlock,
                           AreaReady := "Room2_AreaReady",
                           BeamAllowed := "Room2_BeamAllowed",
                           StartAlarm => "Room2_StartAlarm");
END_REGION

REGION Network 4: 管制输出
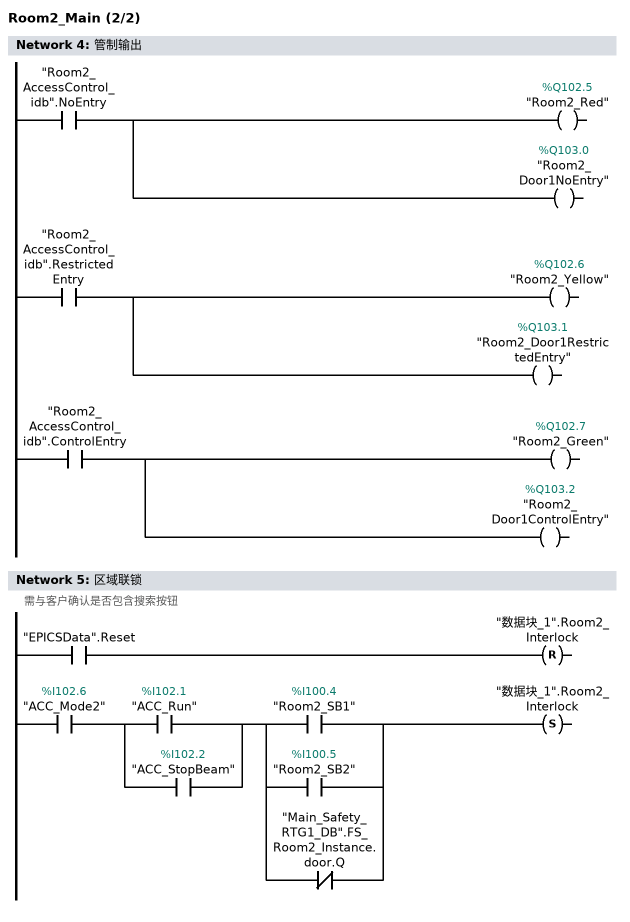
   RUNG wire#powerrail
      Contact( "Room2_AccessControl_idb".NoEntry )
      wire#w1
      Coil( "Room2_Red" )
   END_RUNG
   RUNG wire#w1
      Coil( "Room2_Door1NoEntry" )
   END_RUNG
   RUNG wire#powerrail
      Contact( "Room2_AccessControl_idb".RestrictedEntry )
      wire#w2
      Coil( "Room2_Yellow" )
   END_RUNG
   RUNG wire#w2
      Coil( "Room2_Door1RestrictedEntry" )
   END_RUNG
   RUNG wire#powerrail
      Contact( "Room2_AccessControl_idb".ControlEntry )
      wire#w3
      Coil( "Room2_Green" )
   END_RUNG
   RUNG wire#w3
      Coil( "Room2_Door1ControlEntry" )
   END_RUNG
   // the same network as SCL:
   "Room2_Red" := "Room2_AccessControl_idb".NoEntry;
   "Room2_Door1NoEntry" := "Room2_AccessControl_idb".NoEntry;
   "Room2_Yellow" := "Room2_AccessControl_idb".RestrictedEntry;
   "Room2_Door1RestrictedEntry" := "Room2_AccessControl_idb".RestrictedEntry;
   "Room2_Green" := "Room2_AccessControl_idb".ControlEntry;
   "Room2_Door1ControlEntry" := "Room2_AccessControl_idb".ControlEntry;
END_REGION

REGION Network 5: 区域联锁
   // 需与客户确认是否包含搜索按钮
   RUNG wire#powerrail
      Contact( "EPICSData".Reset )
      R_Coil( "数据块_1".Room2_Interlock )
   END_RUNG
   RUNG wire#powerrail
      Contact( "ACC_Mode2" )
      wire#w1
      Contact( "ACC_Run" )
      wire#w2
      Contact( "Room2_SB1" )
      wire#w3
      S_Coil( "数据块_1".Room2_Interlock )
   END_RUNG
   RUNG wire#w1
      Contact( "ACC_StopBeam" )
   END_RUNG wire#w2
   RUNG wire#w2
      Contact( "Room2_SB2" )
   END_RUNG wire#w3
   RUNG wire#w2
      I_Contact( "Main_Safety_RTG1_DB".FS_Room2_Instance.door.Q )
   END_RUNG wire#w3
   // the same network as SCL:
   IF "EPICSData".Reset THEN "数据块_1".Room2_Interlock := FALSE; END_IF;
   IF "ACC_Mode2" AND ("ACC_Run" OR "ACC_StopBeam") AND ("Room2_SB1" OR "Room2_SB2" OR NOT "Main_Safety_RTG1_DB".FS_Room2_Instance.door.Q) THEN
       "数据块_1".Room2_Interlock := TRUE;
   END_IF;
END_REGION
END_FUNCTION

FUNCTION "ACC_Main" : Void   // FC6, LAD
{ S7_Optimized_Access := 'TRUE' }
VERSION : 0.1
// stored: AutoNumber true, IsIECCheckEnabled false, SetENOAutomatically false, UDAEnableTagReadback false
BEGIN

REGION Network 1: 区域搜索
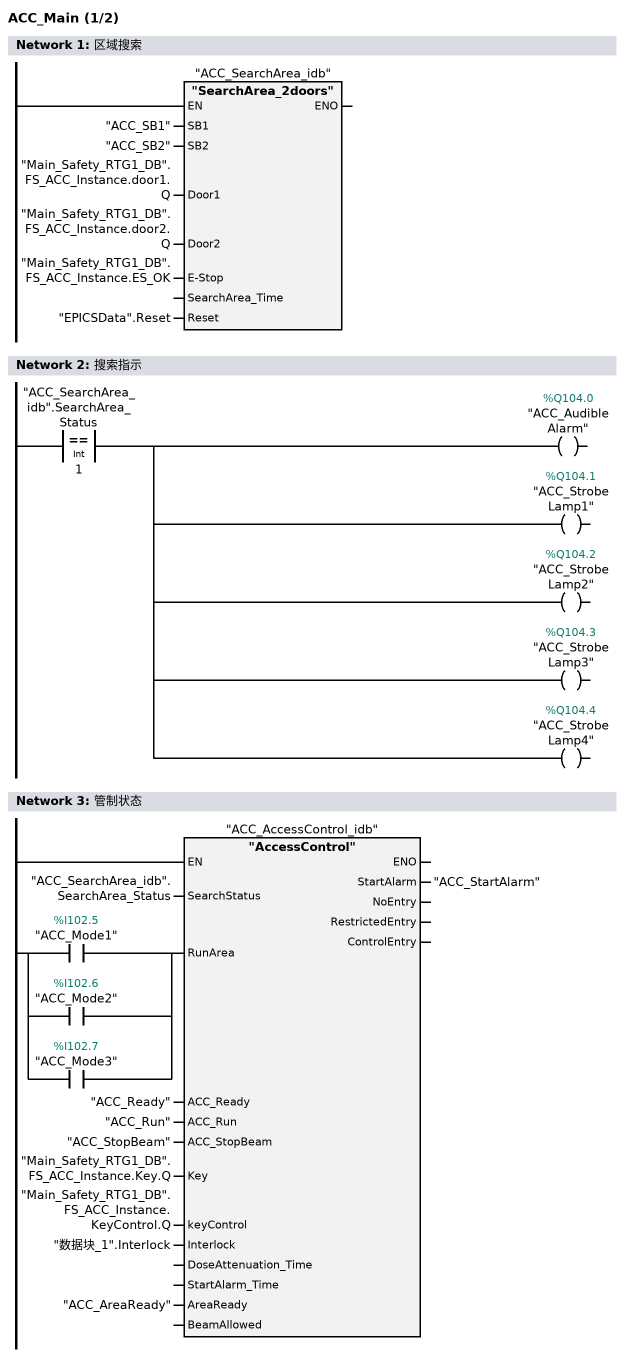
   RUNG wire#powerrail
      "ACC_SearchArea_idb"(SB1 := "ACC_SB1", SB2 := "ACC_SB2", Door1 := "Main_Safety_RTG1_DB".FS_ACC_Instance.door1.Q, Door2 := "Main_Safety_RTG1_DB".FS_ACC_Instance.door2.Q, "E-Stop" := "Main_Safety_RTG1_DB".FS_ACC_Instance.ES_OK, SearchArea_Time :=, Reset := "EPICSData".Reset)
   END_RUNG
   // the same network as SCL:
   "ACC_SearchArea_idb"(SB1 := "ACC_SB1",   // "SearchArea_2doors"
                        SB2 := "ACC_SB2",
                        Door1 := "Main_Safety_RTG1_DB".FS_ACC_Instance.door1.Q,
                        Door2 := "Main_Safety_RTG1_DB".FS_ACC_Instance.door2.Q,
                        "E-Stop" := "Main_Safety_RTG1_DB".FS_ACC_Instance.ES_OK,
                        Reset := "EPICSData".Reset);
END_REGION

REGION Network 2: 搜索指示
   RUNG wire#powerrail
      { S7_Templates := "SrcType := Int" } EQ_Contact(in1 := "ACC_SearchArea_idb".SearchArea_Status, in2 := 1)
      wire#w1
      Coil( "ACC_AudibleAlarm" )
   END_RUNG
   RUNG wire#w1
      Coil( "ACC_StrobeLamp1" )
   END_RUNG
   RUNG wire#w1
      Coil( "ACC_StrobeLamp2" )
   END_RUNG
   RUNG wire#w1
      Coil( "ACC_StrobeLamp3" )
   END_RUNG
   RUNG wire#w1
      Coil( "ACC_StrobeLamp4" )
   END_RUNG
   // the same network as SCL:
   "ACC_AudibleAlarm" := "ACC_SearchArea_idb".SearchArea_Status = 1;
   "ACC_StrobeLamp1" := "ACC_AudibleAlarm";
   "ACC_StrobeLamp2" := "ACC_AudibleAlarm";
   "ACC_StrobeLamp3" := "ACC_AudibleAlarm";
   "ACC_StrobeLamp4" := "ACC_AudibleAlarm";
END_REGION

REGION Network 3: 管制状态
   RUNG wire#powerrail
      "ACC_AccessControl_idb"(RunArea := wire#w1, SearchStatus := "ACC_SearchArea_idb".SearchArea_Status, ACC_Ready := "ACC_Ready", ACC_Run := "ACC_Run", ACC_StopBeam := "ACC_StopBeam", Key := "Main_Safety_RTG1_DB".FS_ACC_Instance.Key.Q, keyControl := "Main_Safety_RTG1_DB".FS_ACC_Instance.KeyControl.Q, Interlock := "数据块_1".Interlock, DoseAttenuation_Time :=, StartAlarm_Time :=, AreaReady := "ACC_AreaReady", BeamAllowed :=, StartAlarm => "ACC_StartAlarm", NoEntry =>, RestrictedEntry =>, ControlEntry =>)
   END_RUNG
   RUNG wire#powerrail
      Contact( "ACC_Mode1" )
   END_RUNG wire#w1
   RUNG wire#powerrail
      Contact( "ACC_Mode2" )
   END_RUNG wire#w1
   RUNG wire#powerrail
      Contact( "ACC_Mode3" )
   END_RUNG wire#w1
   // the same network as SCL:
   "ACC_AccessControl_idb"(SearchStatus := "ACC_SearchArea_idb".SearchArea_Status,   // "AccessControl"
                           RunArea := "ACC_Mode1" OR "ACC_Mode2" OR "ACC_Mode3",
                           ACC_Ready := "ACC_Ready",
                           ACC_Run := "ACC_Run",
                           ACC_StopBeam := "ACC_StopBeam",
                           Key := "Main_Safety_RTG1_DB".FS_ACC_Instance.Key.Q,
                           keyControl := "Main_Safety_RTG1_DB".FS_ACC_Instance.KeyControl.Q,
                           Interlock := "数据块_1".Interlock,
                           AreaReady := "ACC_AreaReady",
                           StartAlarm => "ACC_StartAlarm");
END_REGION

REGION Network 4: 管制输出
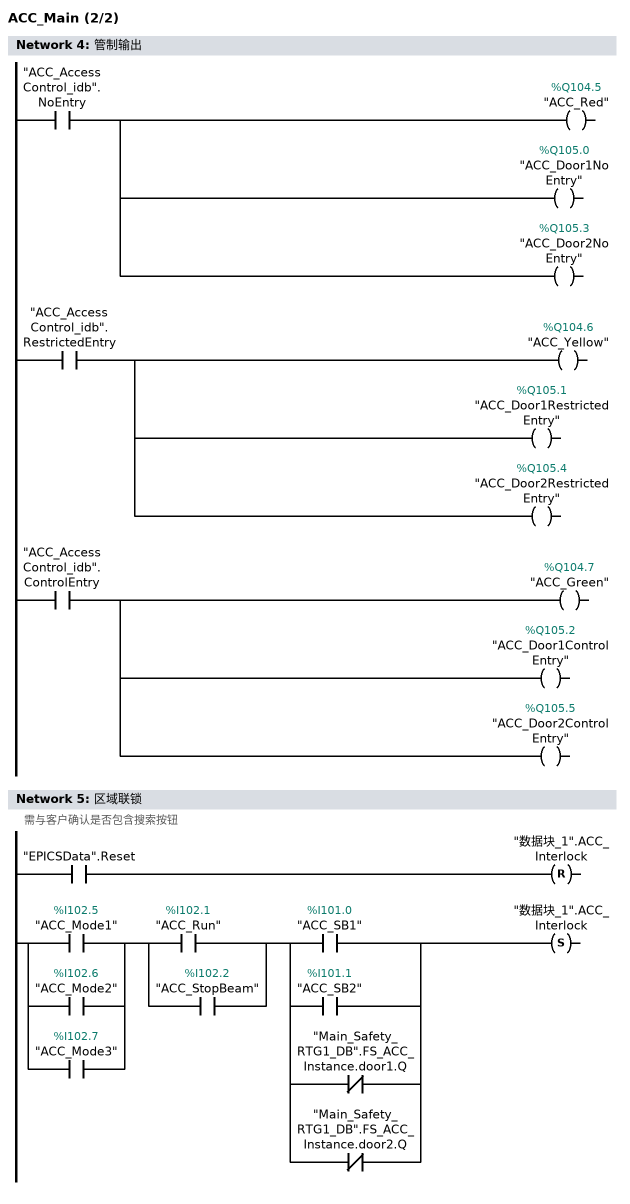
   RUNG wire#powerrail
      Contact( "ACC_AccessControl_idb".NoEntry )
      wire#w1
      Coil( "ACC_Red" )
   END_RUNG
   RUNG wire#w1
      Coil( "ACC_Door1NoEntry" )
   END_RUNG
   RUNG wire#w1
      Coil( "ACC_Door2NoEntry" )
   END_RUNG
   RUNG wire#powerrail
      Contact( "ACC_AccessControl_idb".RestrictedEntry )
      wire#w2
      Coil( "ACC_Yellow" )
   END_RUNG
   RUNG wire#w2
      Coil( "ACC_Door1RestrictedEntry" )
   END_RUNG
   RUNG wire#w2
      Coil( "ACC_Door2RestrictedEntry" )
   END_RUNG
   RUNG wire#powerrail
      Contact( "ACC_AccessControl_idb".ControlEntry )
      wire#w3
      Coil( "ACC_Green" )
   END_RUNG
   RUNG wire#w3
      Coil( "ACC_Door1ControlEntry" )
   END_RUNG
   RUNG wire#w3
      Coil( "ACC_Door2ControlEntry" )
   END_RUNG
   // the same network as SCL:
   "ACC_Red" := "ACC_AccessControl_idb".NoEntry;
   "ACC_Door1NoEntry" := "ACC_AccessControl_idb".NoEntry;
   "ACC_Door2NoEntry" := "ACC_AccessControl_idb".NoEntry;
   "ACC_Yellow" := "ACC_AccessControl_idb".RestrictedEntry;
   "ACC_Door1RestrictedEntry" := "ACC_AccessControl_idb".RestrictedEntry;
   "ACC_Door2RestrictedEntry" := "ACC_AccessControl_idb".RestrictedEntry;
   "ACC_Green" := "ACC_AccessControl_idb".ControlEntry;
   "ACC_Door1ControlEntry" := "ACC_AccessControl_idb".ControlEntry;
   "ACC_Door2ControlEntry" := "ACC_AccessControl_idb".ControlEntry;
END_REGION

REGION Network 5: 区域联锁
   // 需与客户确认是否包含搜索按钮
   RUNG wire#powerrail
      Contact( "EPICSData".Reset )
      R_Coil( "数据块_1".ACC_Interlock )
   END_RUNG
   RUNG wire#powerrail
      Contact( "ACC_Mode1" )
      wire#w1
      Contact( "ACC_Run" )
      wire#w2
      Contact( "ACC_SB1" )
      wire#w3
      S_Coil( "数据块_1".ACC_Interlock )
   END_RUNG
   RUNG wire#powerrail
      Contact( "ACC_Mode2" )
   END_RUNG wire#w1
   RUNG wire#powerrail
      Contact( "ACC_Mode3" )
   END_RUNG wire#w1
   RUNG wire#w1
      Contact( "ACC_StopBeam" )
   END_RUNG wire#w2
   RUNG wire#w2
      Contact( "ACC_SB2" )
   END_RUNG wire#w3
   RUNG wire#w2
      I_Contact( "Main_Safety_RTG1_DB".FS_ACC_Instance.door1.Q )
   END_RUNG wire#w3
   RUNG wire#w2
      I_Contact( "Main_Safety_RTG1_DB".FS_ACC_Instance.door2.Q )
   END_RUNG wire#w3
   // the same network as SCL:
   IF "EPICSData".Reset THEN "数据块_1".ACC_Interlock := FALSE; END_IF;
   IF ("ACC_Mode1" OR "ACC_Mode2" OR "ACC_Mode3") AND ("ACC_Run" OR "ACC_StopBeam") AND ("ACC_SB1" OR "ACC_SB2" OR NOT "Main_Safety_RTG1_DB".FS_ACC_Instance.door1.Q OR NOT "Main_Safety_RTG1_DB".FS_ACC_Instance.door2.Q) THEN
       "数据块_1".ACC_Interlock := TRUE;
   END_IF;
END_REGION
END_FUNCTION

FUNCTION_BLOCK "SearchArea_2doors"   // FB8, LAD
{ S7_Optimized_Access := 'TRUE' }
VERSION : 0.1
// stored: AutoNumber true, IsIECCheckEnabled false, IsRetainMemResEnabled false, MemoryReserve 100, SetENOAutomatically false, UDAEnableTagReadback false
   VAR_INPUT
      SB1 : Bool;
      SB2 : Bool;
      Door1 : Bool;
      Door2 : Bool;
      "E-Stop" : Bool;
      SearchArea_Time : Time := T#5m;
      Reset : Bool;
   END_VAR
   VAR
      SearchArea_Timer { S7_SetPoint := 'True'} : TON_TIME;
      SearchArea_Status : Int;   // 0:未搜索;1:搜索中;2:搜索完成;
      "Step" { S7_SetPoint := 'True'} : Int;
      Error { ExternalAccessible := 'False'; ExternalVisible := 'False'; ExternalWritable := 'False'} : Struct
         All { ExternalAccessible := 'False'; ExternalVisible := 'False'; ExternalWritable := 'False'} : Bool;   // 搜索总故障
         StartFail { ExternalAccessible := 'False'; ExternalVisible := 'False'; ExternalWritable := 'False'} : Bool;   // 搜索启动失败，请确认未按下搜索按钮2或未关闭门1或门2
         WrongSequence1 { ExternalAccessible := 'False'; ExternalVisible := 'False'; ExternalWritable := 'False'} : Bool;   // 搜索顺序错误，此时应按下搜索按钮2，请勿按搜索按钮1或关闭门1或门2
         WrongSequence2 { ExternalAccessible := 'False'; ExternalVisible := 'False'; ExternalWritable := 'False'} : Bool;   // 搜索顺序错误，此时应关闭门1，请勿按搜索按钮1或搜索按钮2或门2
         WrongSequence3 { ExternalAccessible := 'False'; ExternalVisible := 'False'; ExternalWritable := 'False'} : Bool;   // 搜索顺序错误，此时应关闭门2，请勿按搜索按钮1或搜索按钮2或打开门1
         Timeout { ExternalAccessible := 'False'; ExternalVisible := 'False'; ExternalWritable := 'False'} : Bool;   // 搜索超时
      END_STRUCT;
   END_VAR
   VAR_TEMP   // added for the SCL form of the ladder/FBD networks
      _w1 : Bool;
   END_VAR
BEGIN

REGION Network 1: 搜索破坏
   // 搜索完成后，当搜索按钮按下，门被打开，急停按钮按下，搜索状态设置为未搜索
   // 需与客户确认破坏条件是否包含搜索按钮和急停？
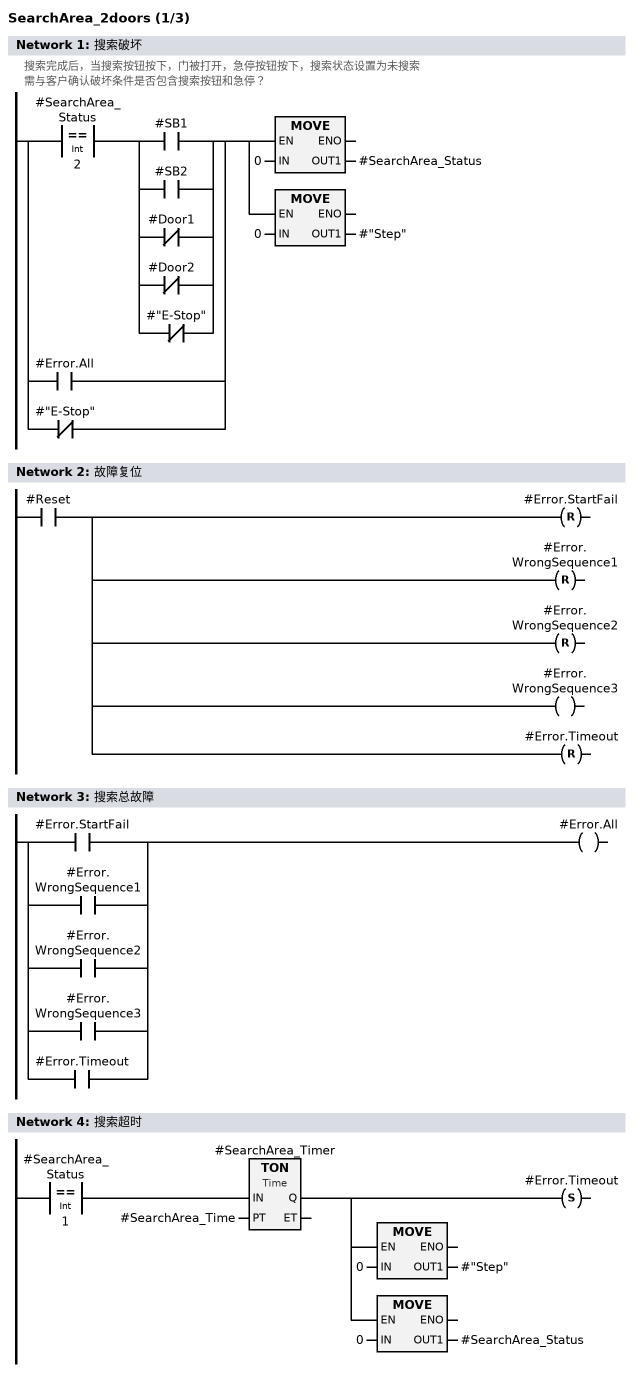
   RUNG wire#powerrail
      { S7_Templates := "SrcType := Int" } EQ_Contact(in1 := #SearchArea_Status, in2 := 2)
      wire#w1
      Contact( #SB1 )
      wire#w2
      Move(in := 0, out1 => #SearchArea_Status)
   END_RUNG
   RUNG wire#w1
      Contact( #SB2 )
   END_RUNG wire#w2
   RUNG wire#w1
      I_Contact( #Door1 )
   END_RUNG wire#w2
   RUNG wire#w1
      I_Contact( #Door2 )
   END_RUNG wire#w2
   RUNG wire#w1
      I_Contact( #"E-Stop" )
   END_RUNG wire#w2
   RUNG wire#powerrail
      Contact( #Error.All )
   END_RUNG wire#w2
   RUNG wire#powerrail
      I_Contact( #"E-Stop" )
   END_RUNG wire#w2
   RUNG wire#w2
      Move(in := 0, out1 => #"Step")
   END_RUNG
   // the same network as SCL:
   #_w1 := ((#SearchArea_Status = 2) AND (#SB1 OR #SB2 OR NOT #Door1 OR NOT #Door2 OR NOT #"E-Stop")) OR #Error.All OR NOT #"E-Stop";
   IF #_w1 THEN
       #SearchArea_Status := 0;
       #"Step" := 0;
   END_IF;
END_REGION

REGION Network 2: 故障复位
   RUNG wire#powerrail
      Contact( #Reset )
      wire#w1
      R_Coil( #Error.StartFail )
   END_RUNG
   RUNG wire#w1
      R_Coil( #Error.WrongSequence1 )
   END_RUNG
   RUNG wire#w1
      R_Coil( #Error.WrongSequence2 )
   END_RUNG
   RUNG wire#w1
      Coil( #Error.WrongSequence3 )
   END_RUNG
   RUNG wire#w1
      R_Coil( #Error.Timeout )
   END_RUNG
   // the same network as SCL:
   IF #Reset THEN
       #Error.StartFail := FALSE;
       #Error.WrongSequence1 := FALSE;
       #Error.WrongSequence2 := FALSE;
   END_IF;
   #Error.WrongSequence3 := #Reset;
   IF #Reset THEN #Error.Timeout := FALSE; END_IF;
END_REGION

REGION Network 3: 搜索总故障
   RUNG wire#powerrail
      Contact( #Error.StartFail )
      wire#w1
      Coil( #Error.All )
   END_RUNG
   RUNG wire#powerrail
      Contact( #Error.WrongSequence1 )
   END_RUNG wire#w1
   RUNG wire#powerrail
      Contact( #Error.WrongSequence2 )
   END_RUNG wire#w1
   RUNG wire#powerrail
      Contact( #Error.WrongSequence3 )
   END_RUNG wire#w1
   RUNG wire#powerrail
      Contact( #Error.Timeout )
   END_RUNG wire#w1
   // the same network as SCL:
   #Error.All := #Error.StartFail OR #Error.WrongSequence1 OR #Error.WrongSequence2 OR #Error.WrongSequence3 OR #Error.Timeout;
END_REGION

REGION Network 4: 搜索超时
   RUNG wire#powerrail
      { S7_Templates := "SrcType := Int" } EQ_Contact(in1 := #SearchArea_Status, in2 := 1)
      { S7_Templates := "time_type := Time" } #SearchArea_Timer.TON(pt := #SearchArea_Time, et =>)
      wire#w1
      S_Coil( #Error.Timeout )
   END_RUNG
   RUNG wire#w1
      Move(in := 0, out1 => #"Step")
   END_RUNG
   RUNG wire#w1
      Move(in := 0, out1 => #SearchArea_Status)
   END_RUNG
   // the same network as SCL:
   #SearchArea_Timer(IN := #SearchArea_Status = 1, PT := #SearchArea_Time);   // TON
   IF #SearchArea_Timer.Q THEN
       #Error.Timeout := TRUE;
       #"Step" := 0;
       #SearchArea_Status := 0;
   END_IF;
END_REGION

REGION Network 5: 按下SB1，开始搜索
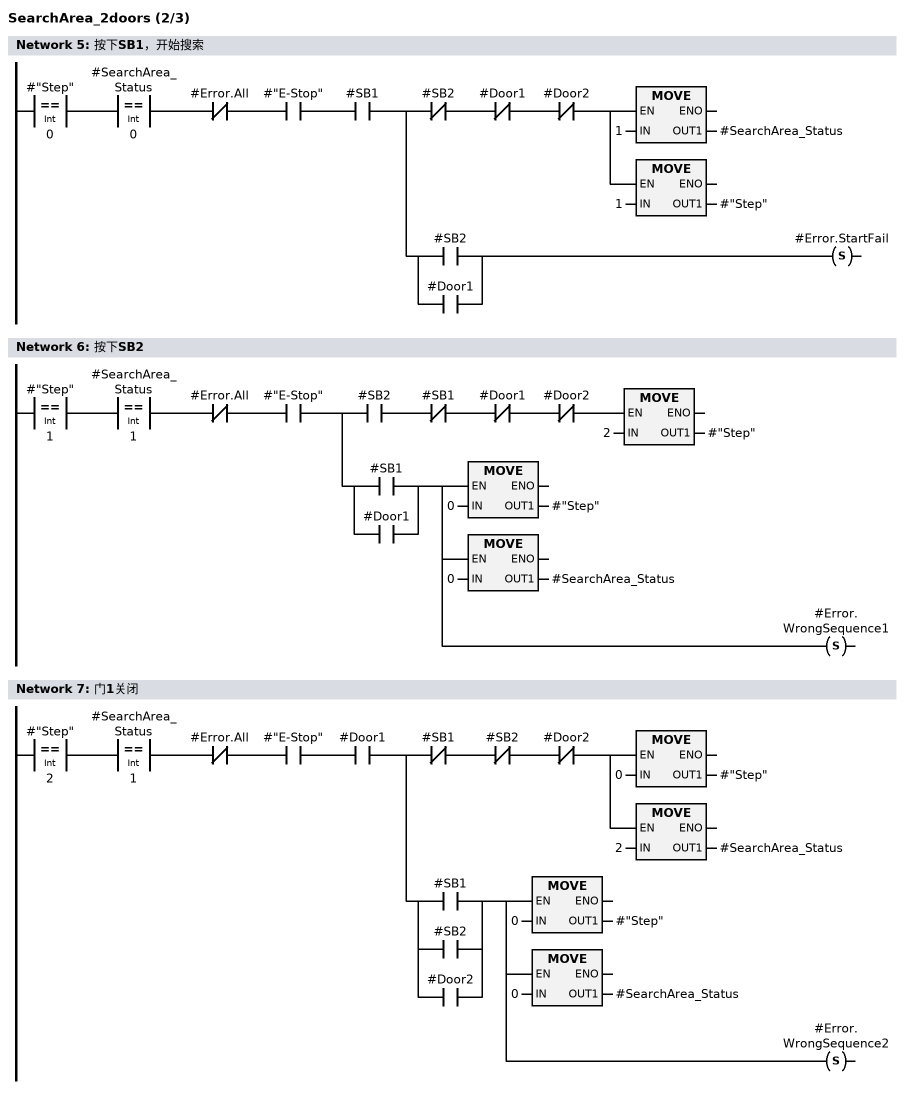
   RUNG wire#powerrail
      { S7_Templates := "SrcType := Int" } EQ_Contact(in1 := #"Step", in2 := 0)
      { S7_Templates := "SrcType := Int" } EQ_Contact(in1 := #SearchArea_Status, in2 := 0)
      I_Contact( #Error.All )
      Contact( #"E-Stop" )
      Contact( #SB1 )
      wire#w1
      I_Contact( #SB2 )
      I_Contact( #Door1 )
      I_Contact( #Door2 )
      wire#w2
      Move(in := 1, out1 => #SearchArea_Status)
   END_RUNG
   RUNG wire#w2
      Move(in := 1, out1 => #"Step")
   END_RUNG
   RUNG wire#w1
      Contact( #SB2 )
      wire#w3
      S_Coil( #Error.StartFail )
   END_RUNG
   RUNG wire#w1
      Contact( #Door1 )
   END_RUNG wire#w3
   // the same network as SCL:
   #_w1 := (#"Step" = 0) AND (#SearchArea_Status = 0) AND NOT #Error.All AND #"E-Stop" AND #SB1;
   IF #_w1 AND NOT #SB2 AND NOT #Door1 AND NOT #Door2 THEN
       #SearchArea_Status := 1;
       #"Step" := 1;
   END_IF;
   IF #_w1 AND (#SB2 OR #Door1) THEN #Error.StartFail := TRUE; END_IF;
END_REGION

REGION Network 6: 按下SB2
   RUNG wire#powerrail
      { S7_Templates := "SrcType := Int" } EQ_Contact(in1 := #"Step", in2 := 1)
      { S7_Templates := "SrcType := Int" } EQ_Contact(in1 := #SearchArea_Status, in2 := 1)
      I_Contact( #Error.All )
      Contact( #"E-Stop" )
      wire#w1
      Contact( #SB2 )
      I_Contact( #SB1 )
      I_Contact( #Door1 )
      I_Contact( #Door2 )
      Move(in := 2, out1 => #"Step")
   END_RUNG
   RUNG wire#w1
      Contact( #SB1 )
      wire#w2
      Move(in := 0, out1 => #"Step")
   END_RUNG
   RUNG wire#w1
      Contact( #Door1 )
   END_RUNG wire#w2
   RUNG wire#w2
      Move(in := 0, out1 => #SearchArea_Status)
   END_RUNG
   RUNG wire#w2
      S_Coil( #Error.WrongSequence1 )
   END_RUNG
   // the same network as SCL:
   #_w1 := (#"Step" = 1) AND (#SearchArea_Status = 1) AND NOT #Error.All AND #"E-Stop";
   IF #_w1 AND #SB2 AND NOT #SB1 AND NOT #Door1 AND NOT #Door2 THEN #"Step" := 2; END_IF;
   IF #_w1 AND (#SB1 OR #Door1) THEN
       #"Step" := 0;
       #SearchArea_Status := 0;
       #Error.WrongSequence1 := TRUE;
   END_IF;
END_REGION

REGION Network 7: 门1关闭
   RUNG wire#powerrail
      { S7_Templates := "SrcType := Int" } EQ_Contact(in1 := #"Step", in2 := 2)
      { S7_Templates := "SrcType := Int" } EQ_Contact(in1 := #SearchArea_Status, in2 := 1)
      I_Contact( #Error.All )
      Contact( #"E-Stop" )
      Contact( #Door1 )
      wire#w1
      I_Contact( #SB1 )
      I_Contact( #SB2 )
      I_Contact( #Door2 )
      wire#w2
      Move(in := 0, out1 => #"Step")
   END_RUNG
   RUNG wire#w2
      Move(in := 2, out1 => #SearchArea_Status)
   END_RUNG
   RUNG wire#w1
      Contact( #SB1 )
      wire#w3
      Move(in := 0, out1 => #"Step")
   END_RUNG
   RUNG wire#w1
      Contact( #SB2 )
   END_RUNG wire#w3
   RUNG wire#w1
      Contact( #Door2 )
   END_RUNG wire#w3
   RUNG wire#w3
      Move(in := 0, out1 => #SearchArea_Status)
   END_RUNG
   RUNG wire#w3
      S_Coil( #Error.WrongSequence2 )
   END_RUNG
   // the same network as SCL:
   #_w1 := (#"Step" = 2) AND (#SearchArea_Status = 1) AND NOT #Error.All AND #"E-Stop" AND #Door1;
   IF #_w1 AND NOT #SB1 AND NOT #SB2 AND NOT #Door2 THEN
       #"Step" := 0;
       #SearchArea_Status := 2;
   END_IF;
   IF #_w1 AND (#SB1 OR #SB2 OR #Door2) THEN
       #"Step" := 0;
       #SearchArea_Status := 0;
       #Error.WrongSequence2 := TRUE;
   END_IF;
END_REGION

REGION Network 8: 门2关闭
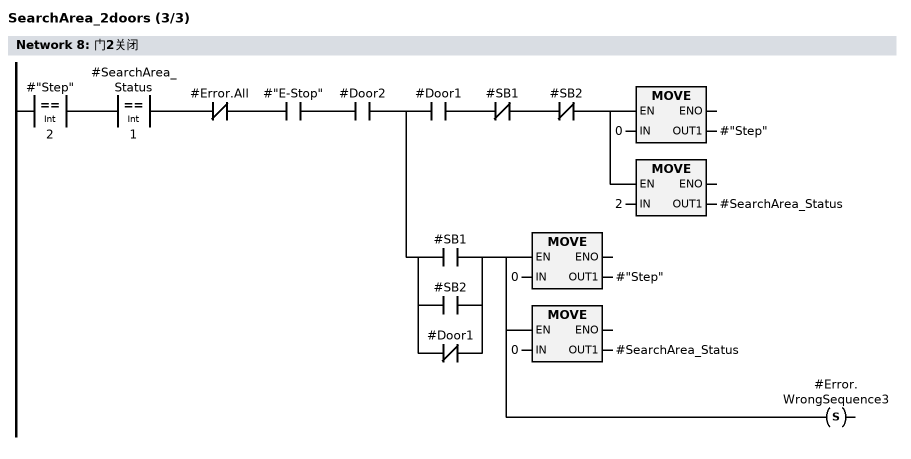
   RUNG wire#powerrail
      { S7_Templates := "SrcType := Int" } EQ_Contact(in1 := #"Step", in2 := 2)
      { S7_Templates := "SrcType := Int" } EQ_Contact(in1 := #SearchArea_Status, in2 := 1)
      I_Contact( #Error.All )
      Contact( #"E-Stop" )
      Contact( #Door2 )
      wire#w1
      Contact( #Door1 )
      I_Contact( #SB1 )
      I_Contact( #SB2 )
      wire#w2
      Move(in := 0, out1 => #"Step")
   END_RUNG
   RUNG wire#w2
      Move(in := 2, out1 => #SearchArea_Status)
   END_RUNG
   RUNG wire#w1
      Contact( #SB1 )
      wire#w3
      Move(in := 0, out1 => #"Step")
   END_RUNG
   RUNG wire#w1
      Contact( #SB2 )
   END_RUNG wire#w3
   RUNG wire#w1
      I_Contact( #Door1 )
   END_RUNG wire#w3
   RUNG wire#w3
      Move(in := 0, out1 => #SearchArea_Status)
   END_RUNG
   RUNG wire#w3
      S_Coil( #Error.WrongSequence3 )
   END_RUNG
   // the same network as SCL:
   #_w1 := (#"Step" = 2) AND (#SearchArea_Status = 1) AND NOT #Error.All AND #"E-Stop" AND #Door2;
   IF #_w1 AND #Door1 AND NOT #SB1 AND NOT #SB2 THEN
       #"Step" := 0;
       #SearchArea_Status := 2;
   END_IF;
   IF #_w1 AND (#SB1 OR #SB2 OR NOT #Door1) THEN
       #"Step" := 0;
       #SearchArea_Status := 0;
       #Error.WrongSequence3 := TRUE;
   END_IF;
END_REGION
END_FUNCTION_BLOCK

FUNCTION "VerticalBeam_Main" : Void   // FC7, LAD
{ S7_Optimized_Access := 'TRUE' }
VERSION : 0.1
// stored: AutoNumber true, IsIECCheckEnabled false, SetENOAutomatically false, UDAEnableTagReadback false
BEGIN

REGION Network 1: 区域搜索
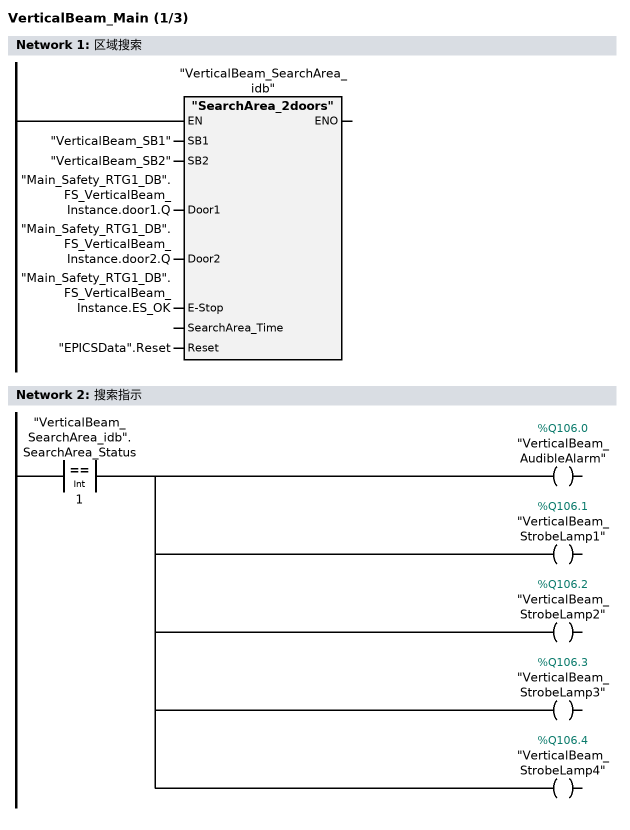
   RUNG wire#powerrail
      "VerticalBeam_SearchArea_idb"(SB1 := "VerticalBeam_SB1", SB2 := "VerticalBeam_SB2", Door1 := "Main_Safety_RTG1_DB".FS_VerticalBeam_Instance.door1.Q, Door2 := "Main_Safety_RTG1_DB".FS_VerticalBeam_Instance.door2.Q, "E-Stop" := "Main_Safety_RTG1_DB".FS_VerticalBeam_Instance.ES_OK, SearchArea_Time :=, Reset := "EPICSData".Reset)
   END_RUNG
   // the same network as SCL:
   "VerticalBeam_SearchArea_idb"(SB1 := "VerticalBeam_SB1",   // "SearchArea_2doors"
                           SB2 := "VerticalBeam_SB2",
                           Door1 := "Main_Safety_RTG1_DB".FS_VerticalBeam_Instance.door1.Q,
                           Door2 := "Main_Safety_RTG1_DB".FS_VerticalBeam_Instance.door2.Q,
                           "E-Stop" := "Main_Safety_RTG1_DB".FS_VerticalBeam_Instance.ES_OK,
                           Reset := "EPICSData".Reset);
END_REGION

REGION Network 2: 搜索指示
   RUNG wire#powerrail
      { S7_Templates := "SrcType := Int" } EQ_Contact(in1 := "VerticalBeam_SearchArea_idb".SearchArea_Status, in2 := 1)
      wire#w1
      Coil( "VerticalBeam_AudibleAlarm" )
   END_RUNG
   RUNG wire#w1
      Coil( "VerticalBeam_StrobeLamp1" )
   END_RUNG
   RUNG wire#w1
      Coil( "VerticalBeam_StrobeLamp2" )
   END_RUNG
   RUNG wire#w1
      Coil( "VerticalBeam_StrobeLamp3" )
   END_RUNG
   RUNG wire#w1
      Coil( "VerticalBeam_StrobeLamp4" )
   END_RUNG
   // the same network as SCL:
   "VerticalBeam_AudibleAlarm" := "VerticalBeam_SearchArea_idb".SearchArea_Status = 1;
   "VerticalBeam_StrobeLamp1" := "VerticalBeam_AudibleAlarm";
   "VerticalBeam_StrobeLamp2" := "VerticalBeam_AudibleAlarm";
   "VerticalBeam_StrobeLamp3" := "VerticalBeam_AudibleAlarm";
   "VerticalBeam_StrobeLamp4" := "VerticalBeam_AudibleAlarm";
END_REGION

REGION Network 3: 管制状态
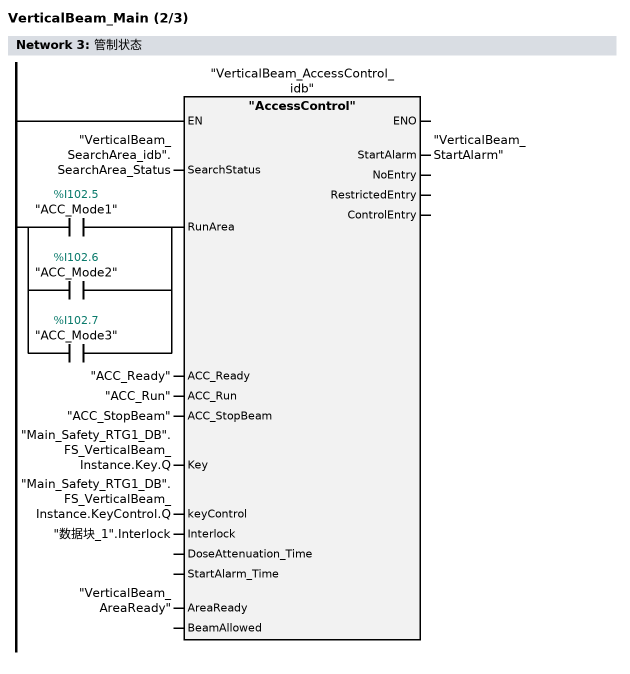
   RUNG wire#powerrail
      "VerticalBeam_AccessControl_idb"(RunArea := wire#w1, SearchStatus := "VerticalBeam_SearchArea_idb".SearchArea_Status, ACC_Ready := "ACC_Ready", ACC_Run := "ACC_Run", ACC_StopBeam := "ACC_StopBeam", Key := "Main_Safety_RTG1_DB".FS_VerticalBeam_Instance.Key.Q, keyControl := "Main_Safety_RTG1_DB".FS_VerticalBeam_Instance.KeyControl.Q, Interlock := "数据块_1".Interlock, DoseAttenuation_Time :=, StartAlarm_Time :=, AreaReady := "VerticalBeam_AreaReady", BeamAllowed :=, StartAlarm => "VerticalBeam_StartAlarm", NoEntry =>, RestrictedEntry =>, ControlEntry =>)
   END_RUNG
   RUNG wire#powerrail
      Contact( "ACC_Mode1" )
   END_RUNG wire#w1
   RUNG wire#powerrail
      Contact( "ACC_Mode2" )
   END_RUNG wire#w1
   RUNG wire#powerrail
      Contact( "ACC_Mode3" )
   END_RUNG wire#w1
   // the same network as SCL:
   "VerticalBeam_AccessControl_idb"(SearchStatus := "VerticalBeam_SearchArea_idb".SearchArea_Status,   // "AccessControl"
                           RunArea := "ACC_Mode1" OR "ACC_Mode2" OR "ACC_Mode3",
                           ACC_Ready := "ACC_Ready",
                           ACC_Run := "ACC_Run",
                           ACC_StopBeam := "ACC_StopBeam",
                           Key := "Main_Safety_RTG1_DB".FS_VerticalBeam_Instance.Key.Q,
                           keyControl := "Main_Safety_RTG1_DB".FS_VerticalBeam_Instance.KeyControl.Q,
                           Interlock := "数据块_1".Interlock,
                           AreaReady := "VerticalBeam_AreaReady",
                           StartAlarm => "VerticalBeam_StartAlarm");
END_REGION

REGION Network 4: 管制输出
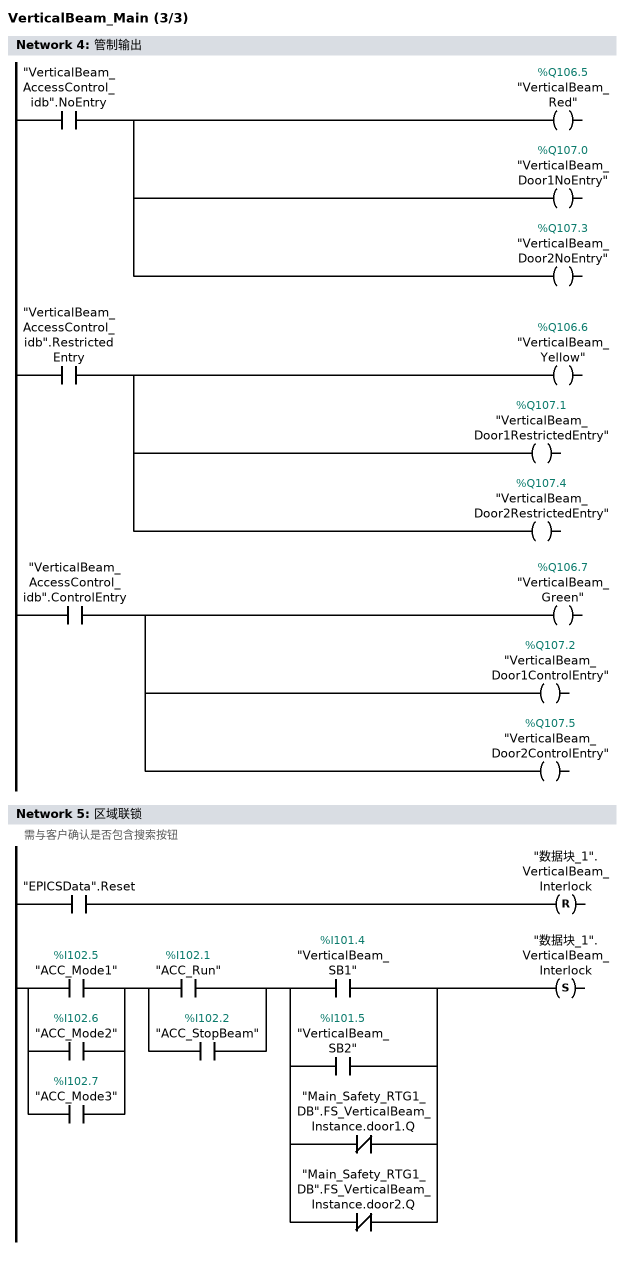
   RUNG wire#powerrail
      Contact( "VerticalBeam_AccessControl_idb".NoEntry )
      wire#w1
      Coil( "VerticalBeam_Red" )
   END_RUNG
   RUNG wire#w1
      Coil( "VerticalBeam_Door1NoEntry" )
   END_RUNG
   RUNG wire#w1
      Coil( "VerticalBeam_Door2NoEntry" )
   END_RUNG
   RUNG wire#powerrail
      Contact( "VerticalBeam_AccessControl_idb".RestrictedEntry )
      wire#w2
      Coil( "VerticalBeam_Yellow" )
   END_RUNG
   RUNG wire#w2
      Coil( "VerticalBeam_Door1RestrictedEntry" )
   END_RUNG
   RUNG wire#w2
      Coil( "VerticalBeam_Door2RestrictedEntry" )
   END_RUNG
   RUNG wire#powerrail
      Contact( "VerticalBeam_AccessControl_idb".ControlEntry )
      wire#w3
      Coil( "VerticalBeam_Green" )
   END_RUNG
   RUNG wire#w3
      Coil( "VerticalBeam_Door1ControlEntry" )
   END_RUNG
   RUNG wire#w3
      Coil( "VerticalBeam_Door2ControlEntry" )
   END_RUNG
   // the same network as SCL:
   "VerticalBeam_Red" := "VerticalBeam_AccessControl_idb".NoEntry;
   "VerticalBeam_Door1NoEntry" := "VerticalBeam_AccessControl_idb".NoEntry;
   "VerticalBeam_Door2NoEntry" := "VerticalBeam_AccessControl_idb".NoEntry;
   "VerticalBeam_Yellow" := "VerticalBeam_AccessControl_idb".RestrictedEntry;
   "VerticalBeam_Door1RestrictedEntry" := "VerticalBeam_AccessControl_idb".RestrictedEntry;
   "VerticalBeam_Door2RestrictedEntry" := "VerticalBeam_AccessControl_idb".RestrictedEntry;
   "VerticalBeam_Green" := "VerticalBeam_AccessControl_idb".ControlEntry;
   "VerticalBeam_Door1ControlEntry" := "VerticalBeam_AccessControl_idb".ControlEntry;
   "VerticalBeam_Door2ControlEntry" := "VerticalBeam_AccessControl_idb".ControlEntry;
END_REGION

REGION Network 5: 区域联锁
   // 需与客户确认是否包含搜索按钮
   RUNG wire#powerrail
      Contact( "EPICSData".Reset )
      R_Coil( "数据块_1".VerticalBeam_Interlock )
   END_RUNG
   RUNG wire#powerrail
      Contact( "ACC_Mode1" )
      wire#w1
      Contact( "ACC_Run" )
      wire#w2
      Contact( "VerticalBeam_SB1" )
      wire#w3
      S_Coil( "数据块_1".VerticalBeam_Interlock )
   END_RUNG
   RUNG wire#powerrail
      Contact( "ACC_Mode2" )
   END_RUNG wire#w1
   RUNG wire#powerrail
      Contact( "ACC_Mode3" )
   END_RUNG wire#w1
   RUNG wire#w1
      Contact( "ACC_StopBeam" )
   END_RUNG wire#w2
   RUNG wire#w2
      Contact( "VerticalBeam_SB2" )
   END_RUNG wire#w3
   RUNG wire#w2
      I_Contact( "Main_Safety_RTG1_DB".FS_VerticalBeam_Instance.door1.Q )
   END_RUNG wire#w3
   RUNG wire#w2
      I_Contact( "Main_Safety_RTG1_DB".FS_VerticalBeam_Instance.door2.Q )
   END_RUNG wire#w3
   // the same network as SCL:
   IF "EPICSData".Reset THEN "数据块_1".VerticalBeam_Interlock := FALSE; END_IF;
   IF ("ACC_Mode1" OR "ACC_Mode2" OR "ACC_Mode3") AND ("ACC_Run" OR "ACC_StopBeam") AND ("VerticalBeam_SB1" OR "VerticalBeam_SB2" OR NOT "Main_Safety_RTG1_DB".FS_VerticalBeam_Instance.door1.Q OR NOT "Main_Safety_RTG1_DB".FS_VerticalBeam_Instance.door2.Q) THEN
       "数据块_1".VerticalBeam_Interlock := TRUE;
   END_IF;
END_REGION
END_FUNCTION

ORGANIZATION_BLOCK "Time error interrupt"   // OB80, LAD, TimeErrorInterrupt
{ S7_Optimized_Access := 'TRUE' }
VERSION : 0.1
// stored: IsIECCheckEnabled false, SetENOAutomatically false
   VAR_INPUT
      Fault_ID : Byte;   // Fault identifier
      Csg_OBnr : OB_ANY;   // Number of OB causing the error
      Csg_Prio : UInt;   // Priority of OB causing the error
   END_VAR
BEGIN
END_ORGANIZATION_BLOCK

FUNCTION_BLOCK "FS_ACC"   // FB4, F_LAD
{ S7_Optimized_Access := 'TRUE' }
VERSION : 0.1
// stored: AutoNumber false, IsIECCheckEnabled false, UDAEnableTagReadback false
   VAR_INPUT
      ACK : Bool;
   END_VAR
   VAR_OUTPUT
      ES_OK : Bool;
   END_VAR
   VAR
      EStop1 { S7_SetPoint := 'True'} : ESTOP1;
      EStop2 { S7_SetPoint := 'True'} : ESTOP1;
      EStop3 { S7_SetPoint := 'True'} : ESTOP1;
      EStop4 { S7_SetPoint := 'True'} : ESTOP1;
      door1 : SFDOOR;
      door2 : SFDOOR;
      Key : SFDOOR;
      KeyControl : SFDOOR;
   END_VAR
BEGIN

REGION Network 1: E-Stop1
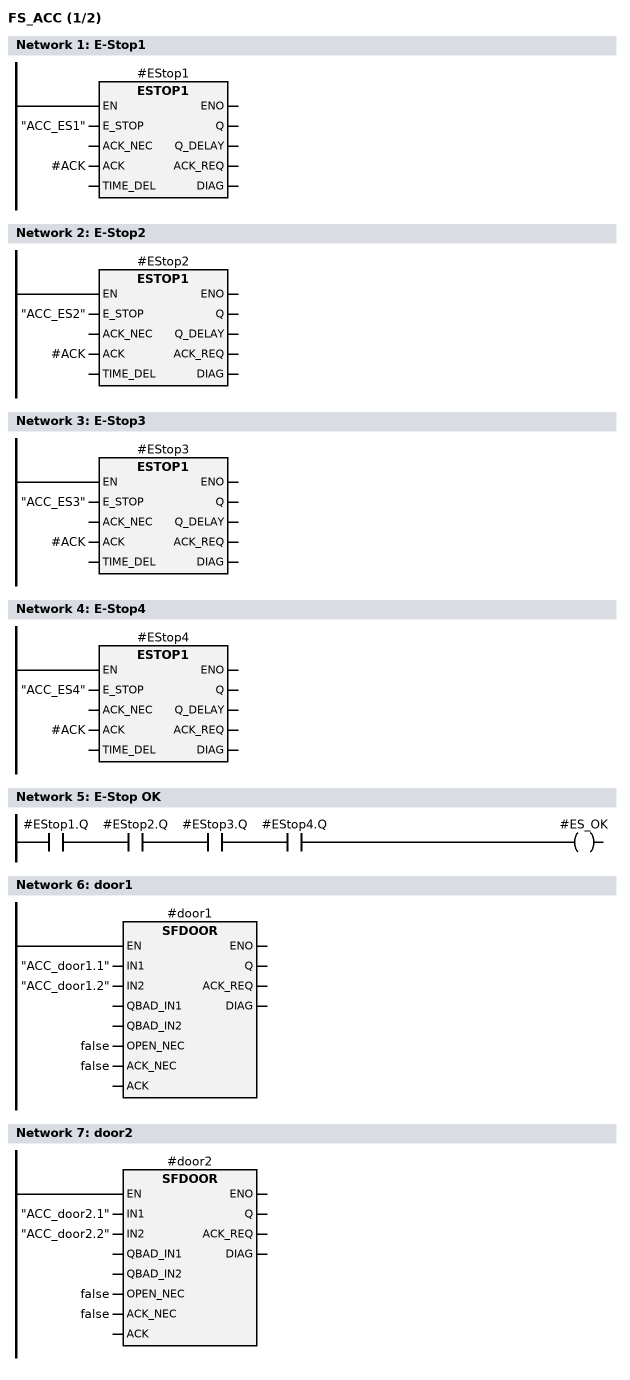
   RUNG wire#powerrail
      #EStop1.ESTOP1(E_STOP := "ACC_ES1", ACK_NEC :=, ACK := #ACK, TIME_DEL :=, Q =>, Q_DELAY =>, ACK_REQ =>, DIAG =>)
   END_RUNG
   // the same network as SCL:
   #EStop1(E_STOP := "ACC_ES1", ACK := #ACK);   // ESTOP1
END_REGION

REGION Network 2: E-Stop2
   RUNG wire#powerrail
      #EStop2.ESTOP1(E_STOP := "ACC_ES2", ACK_NEC :=, ACK := #ACK, TIME_DEL :=, Q =>, Q_DELAY =>, ACK_REQ =>, DIAG =>)
   END_RUNG
   // the same network as SCL:
   #EStop2(E_STOP := "ACC_ES2", ACK := #ACK);   // ESTOP1
END_REGION

REGION Network 3: E-Stop3
   RUNG wire#powerrail
      #EStop3.ESTOP1(E_STOP := "ACC_ES3", ACK_NEC :=, ACK := #ACK, TIME_DEL :=, Q =>, Q_DELAY =>, ACK_REQ =>, DIAG =>)
   END_RUNG
   // the same network as SCL:
   #EStop3(E_STOP := "ACC_ES3", ACK := #ACK);   // ESTOP1
END_REGION

REGION Network 4: E-Stop4
   RUNG wire#powerrail
      #EStop4.ESTOP1(E_STOP := "ACC_ES4", ACK_NEC :=, ACK := #ACK, TIME_DEL :=, Q =>, Q_DELAY =>, ACK_REQ =>, DIAG =>)
   END_RUNG
   // the same network as SCL:
   #EStop4(E_STOP := "ACC_ES4", ACK := #ACK);   // ESTOP1
END_REGION

REGION Network 5: E-Stop OK
   RUNG wire#powerrail
      Contact( #EStop1.Q )
      Contact( #EStop2.Q )
      Contact( #EStop3.Q )
      Contact( #EStop4.Q )
      Coil( #ES_OK )
   END_RUNG
   // the same network as SCL:
   #ES_OK := #EStop1.Q AND #EStop2.Q AND #EStop3.Q AND #EStop4.Q;
END_REGION

REGION Network 6: door1
   RUNG wire#powerrail
      #door1.SFDOOR(IN1 := "ACC_door1.1", IN2 := "ACC_door1.2", QBAD_IN1 :=, QBAD_IN2 :=, OPEN_NEC := false, ACK_NEC := false, ACK :=, Q =>, ACK_REQ =>, DIAG =>)
   END_RUNG
   // the same network as SCL:
   #door1(IN1 := "ACC_door1.1", IN2 := "ACC_door1.2", OPEN_NEC := false, ACK_NEC := false);   // SFDOOR
END_REGION

REGION Network 7: door2
   RUNG wire#powerrail
      #door2.SFDOOR(IN1 := "ACC_door2.1", IN2 := "ACC_door2.2", QBAD_IN1 :=, QBAD_IN2 :=, OPEN_NEC := false, ACK_NEC := false, ACK :=, Q =>, ACK_REQ =>, DIAG =>)
   END_RUNG
   // the same network as SCL:
   #door2(IN1 := "ACC_door2.1", IN2 := "ACC_door2.2", OPEN_NEC := false, ACK_NEC := false);   // SFDOOR
END_REGION

REGION Network 8: Key
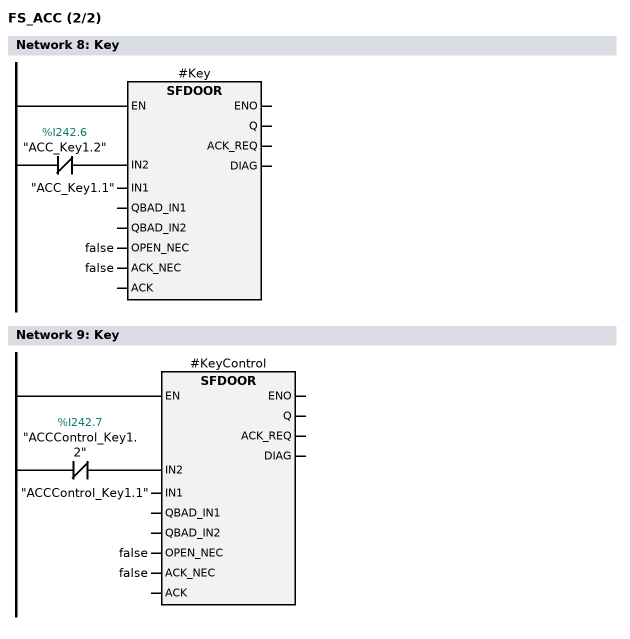
   RUNG wire#powerrail
      #Key.SFDOOR(IN2 := wire#w1, IN1 := "ACC_Key1.1", QBAD_IN1 :=, QBAD_IN2 :=, OPEN_NEC := false, ACK_NEC := false, ACK :=, Q =>, ACK_REQ =>, DIAG =>)
   END_RUNG
   RUNG wire#powerrail
      I_Contact( "ACC_Key1.2" )
   END_RUNG wire#w1
   // the same network as SCL:
   #Key(IN2 := NOT "ACC_Key1.2", IN1 := "ACC_Key1.1", OPEN_NEC := false, ACK_NEC := false);   // SFDOOR
END_REGION

REGION Network 9: Key
   RUNG wire#powerrail
      #KeyControl.SFDOOR(IN2 := wire#w1, IN1 := "ACCControl_Key1.1", QBAD_IN1 :=, QBAD_IN2 :=, OPEN_NEC := false, ACK_NEC := false, ACK :=, Q =>, ACK_REQ =>, DIAG =>)
   END_RUNG
   RUNG wire#powerrail
      I_Contact( "ACCControl_Key1.2" )
   END_RUNG wire#w1
   // the same network as SCL:
   #KeyControl(IN2 := NOT "ACCControl_Key1.2", IN1 := "ACCControl_Key1.1", OPEN_NEC := false, ACK_NEC := false);   // SFDOOR
END_REGION
END_FUNCTION_BLOCK

FUNCTION_BLOCK "FS_Room1"   // FB2, F_LAD
{ S7_Optimized_Access := 'TRUE' }
VERSION : 0.1
// 急停：2NC 硬件组态配置
// 1,急停故障
// 2,急停已恢复，需要确认
// 
// 
// 钥匙：1NC+1NO
// 1，钥匙电磁基座信号不匹配
// 2，基座信号正常，需要确认
// 3，安全钥匙2个电磁基座信号一致性故障，均显示插入
// 4，安全钥匙2个电磁基座信号一致性正常，需要确认
// 
// 门：2NC时关闭
// 1，门信号不一致，需要同时开同时关闭
// stored: AutoNumber true, IsIECCheckEnabled false, UDAEnableTagReadback false
   VAR_INPUT
      ACK : Bool;
   END_VAR
   VAR_OUTPUT
      ES_OK : Bool;
   END_VAR
   VAR
      EStop1 { S7_SetPoint := 'True'} : ESTOP1;
      EStop2 { S7_SetPoint := 'True'} : ESTOP1;
      EStop3 { S7_SetPoint := 'True'} : ESTOP1;
      EStop4 { S7_SetPoint := 'True'} : ESTOP1;
      EStop5 { S7_SetPoint := 'True'} : ESTOP1;
      EStop6 : ESTOP1;
      door : SFDOOR;
      Key : SFDOOR;
      KeyControl : SFDOOR;
      Door_Timer : TON;
      Key1 : TON;
      KeyControl1 : TON;
      Key_InDoor : Bool;
      Key_InControl : Bool;
   END_VAR
BEGIN

REGION Network 1: E-Stop1
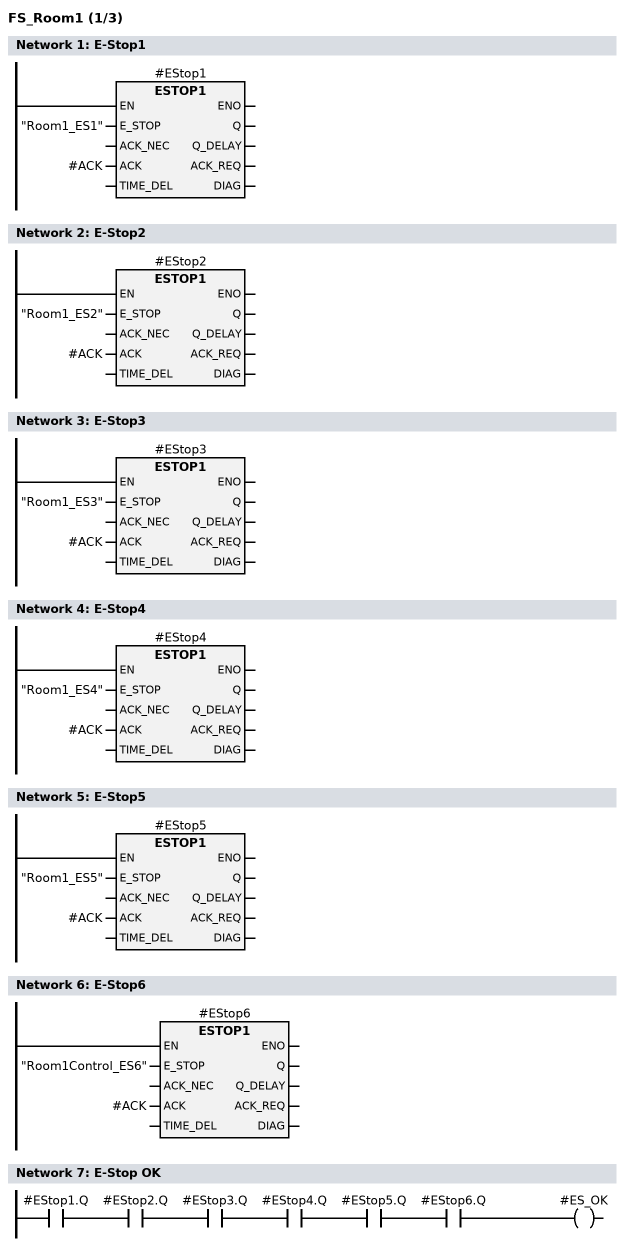
   RUNG wire#powerrail
      #EStop1.ESTOP1(E_STOP := "Room1_ES1", ACK_NEC :=, ACK := #ACK, TIME_DEL :=, Q =>, Q_DELAY =>, ACK_REQ =>, DIAG =>)
   END_RUNG
   // the same network as SCL:
   #EStop1(E_STOP := "Room1_ES1", ACK := #ACK);   // ESTOP1
END_REGION

REGION Network 2: E-Stop2
   RUNG wire#powerrail
      #EStop2.ESTOP1(E_STOP := "Room1_ES2", ACK_NEC :=, ACK := #ACK, TIME_DEL :=, Q =>, Q_DELAY =>, ACK_REQ =>, DIAG =>)
   END_RUNG
   // the same network as SCL:
   #EStop2(E_STOP := "Room1_ES2", ACK := #ACK);   // ESTOP1
END_REGION

REGION Network 3: E-Stop3
   RUNG wire#powerrail
      #EStop3.ESTOP1(E_STOP := "Room1_ES3", ACK_NEC :=, ACK := #ACK, TIME_DEL :=, Q =>, Q_DELAY =>, ACK_REQ =>, DIAG =>)
   END_RUNG
   // the same network as SCL:
   #EStop3(E_STOP := "Room1_ES3", ACK := #ACK);   // ESTOP1
END_REGION

REGION Network 4: E-Stop4
   RUNG wire#powerrail
      #EStop4.ESTOP1(E_STOP := "Room1_ES4", ACK_NEC :=, ACK := #ACK, TIME_DEL :=, Q =>, Q_DELAY =>, ACK_REQ =>, DIAG =>)
   END_RUNG
   // the same network as SCL:
   #EStop4(E_STOP := "Room1_ES4", ACK := #ACK);   // ESTOP1
END_REGION

REGION Network 5: E-Stop5
   RUNG wire#powerrail
      #EStop5.ESTOP1(E_STOP := "Room1_ES5", ACK_NEC :=, ACK := #ACK, TIME_DEL :=, Q =>, Q_DELAY =>, ACK_REQ =>, DIAG =>)
   END_RUNG
   // the same network as SCL:
   #EStop5(E_STOP := "Room1_ES5", ACK := #ACK);   // ESTOP1
END_REGION

REGION Network 6: E-Stop6
   RUNG wire#powerrail
      #EStop6.ESTOP1(E_STOP := "Room1Control_ES6", ACK_NEC :=, ACK := #ACK, TIME_DEL :=, Q =>, Q_DELAY =>, ACK_REQ =>, DIAG =>)
   END_RUNG
   // the same network as SCL:
   #EStop6(E_STOP := "Room1Control_ES6", ACK := #ACK);   // ESTOP1
END_REGION

REGION Network 7: E-Stop OK
   RUNG wire#powerrail
      Contact( #EStop1.Q )
      Contact( #EStop2.Q )
      Contact( #EStop3.Q )
      Contact( #EStop4.Q )
      Contact( #EStop5.Q )
      Contact( #EStop6.Q )
      Coil( #ES_OK )
   END_RUNG
   // the same network as SCL:
   #ES_OK := #EStop1.Q AND #EStop2.Q AND #EStop3.Q AND #EStop4.Q AND #EStop5.Q AND #EStop6.Q;
END_REGION

REGION Network 8: door
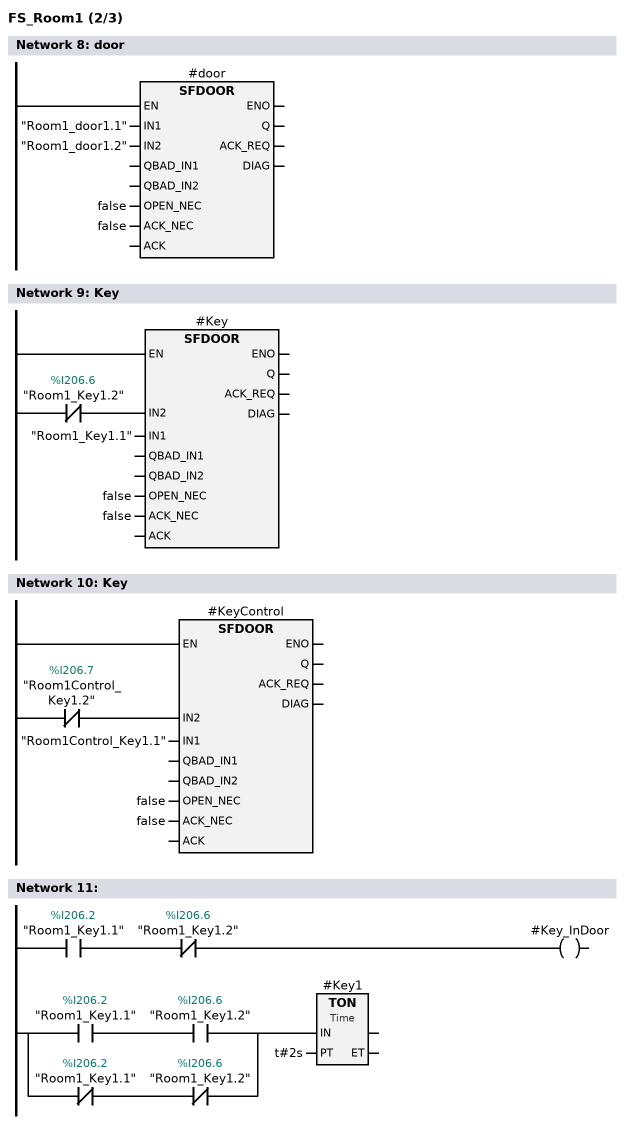
   RUNG wire#powerrail
      #door.SFDOOR(IN1 := "Room1_door1.1", IN2 := "Room1_door1.2", QBAD_IN1 :=, QBAD_IN2 :=, OPEN_NEC := false, ACK_NEC := false, ACK :=, Q =>, ACK_REQ =>, DIAG =>)
   END_RUNG
   // the same network as SCL:
   #door(IN1 := "Room1_door1.1", IN2 := "Room1_door1.2", OPEN_NEC := false, ACK_NEC := false);   // SFDOOR
END_REGION

REGION Network 9: Key
   RUNG wire#powerrail
      #Key.SFDOOR(IN2 := wire#w1, IN1 := "Room1_Key1.1", QBAD_IN1 :=, QBAD_IN2 :=, OPEN_NEC := false, ACK_NEC := false, ACK :=, Q =>, ACK_REQ =>, DIAG =>)
   END_RUNG
   RUNG wire#powerrail
      I_Contact( "Room1_Key1.2" )
   END_RUNG wire#w1
   // the same network as SCL:
   #Key(IN2 := NOT "Room1_Key1.2", IN1 := "Room1_Key1.1", OPEN_NEC := false, ACK_NEC := false);   // SFDOOR
END_REGION

REGION Network 10: Key
   RUNG wire#powerrail
      #KeyControl.SFDOOR(IN2 := wire#w1, IN1 := "Room1Control_Key1.1", QBAD_IN1 :=, QBAD_IN2 :=, OPEN_NEC := false, ACK_NEC := false, ACK :=, Q =>, ACK_REQ =>, DIAG =>)
   END_RUNG
   RUNG wire#powerrail
      I_Contact( "Room1Control_Key1.2" )
   END_RUNG wire#w1
   // the same network as SCL:
   #KeyControl(IN2 := NOT "Room1Control_Key1.2",   // SFDOOR
               IN1 := "Room1Control_Key1.1",
               OPEN_NEC := false,
               ACK_NEC := false);
END_REGION

REGION Network 11
   RUNG wire#powerrail
      Contact( "Room1_Key1.1" )
      I_Contact( "Room1_Key1.2" )
      Coil( #Key_InDoor )
   END_RUNG
   RUNG wire#powerrail
      Contact( "Room1_Key1.1" )
      Contact( "Room1_Key1.2" )
      wire#w1
      { S7_Templates := "[time_type := Time, codedbool_type := DInt]" } #Key1.TON(pt := t#2s, et =>)
   END_RUNG
   RUNG wire#powerrail
      I_Contact( "Room1_Key1.1" )
      I_Contact( "Room1_Key1.2" )
   END_RUNG wire#w1
   // the same network as SCL:
   #Key_InDoor := "Room1_Key1.1" AND NOT "Room1_Key1.2";
   #Key1.TON(IN := ("Room1_Key1.1" AND "Room1_Key1.2") OR (NOT "Room1_Key1.1" AND NOT "Room1_Key1.2"),
             PT := t#2s);
END_REGION

REGION Network 12
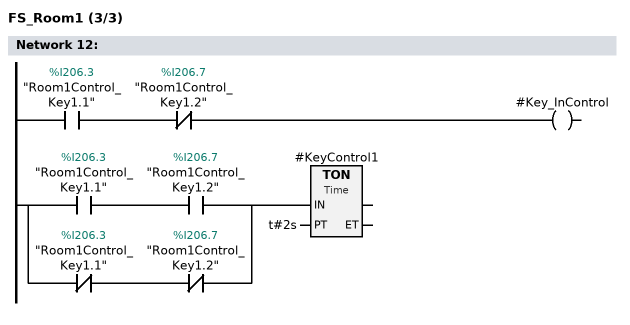
   RUNG wire#powerrail
      Contact( "Room1Control_Key1.1" )
      I_Contact( "Room1Control_Key1.2" )
      Coil( #Key_InControl )
   END_RUNG
   RUNG wire#powerrail
      Contact( "Room1Control_Key1.1" )
      Contact( "Room1Control_Key1.2" )
      wire#w1
      { S7_Templates := "[time_type := Time, codedbool_type := DInt]" } #KeyControl1.TON(pt := t#2s, et =>)
   END_RUNG
   RUNG wire#powerrail
      I_Contact( "Room1Control_Key1.1" )
      I_Contact( "Room1Control_Key1.2" )
   END_RUNG wire#w1
   // the same network as SCL:
   #Key_InControl := "Room1Control_Key1.1" AND NOT "Room1Control_Key1.2";
   #KeyControl1.TON(IN := ("Room1Control_Key1.1" AND "Room1Control_Key1.2") OR (NOT "Room1Control_Key1.1" AND NOT "Room1Control_Key1.2"),
                    PT := t#2s);
END_REGION
END_FUNCTION_BLOCK

FUNCTION_BLOCK "FS_Room2"   // FB3, F_LAD
{ S7_Optimized_Access := 'TRUE' }
VERSION : 0.1
// stored: AutoNumber false, IsIECCheckEnabled false, UDAEnableTagReadback false
   VAR_INPUT
      ACK : Bool;
   END_VAR
   VAR_OUTPUT
      ES_OK : Bool;
   END_VAR
   VAR
      EStop1 { S7_SetPoint := 'True'} : ESTOP1;
      EStop2 { S7_SetPoint := 'True'} : ESTOP1;
      EStop3 { S7_SetPoint := 'True'} : ESTOP1;
      EStop4 { S7_SetPoint := 'True'} : ESTOP1;
      EStop5 { S7_SetPoint := 'True'} : ESTOP1;
      EStop6 : ESTOP1;
      door : SFDOOR;
      Key : SFDOOR;
      KeyControl : SFDOOR;
   END_VAR
BEGIN

REGION Network 1: E-Stop1
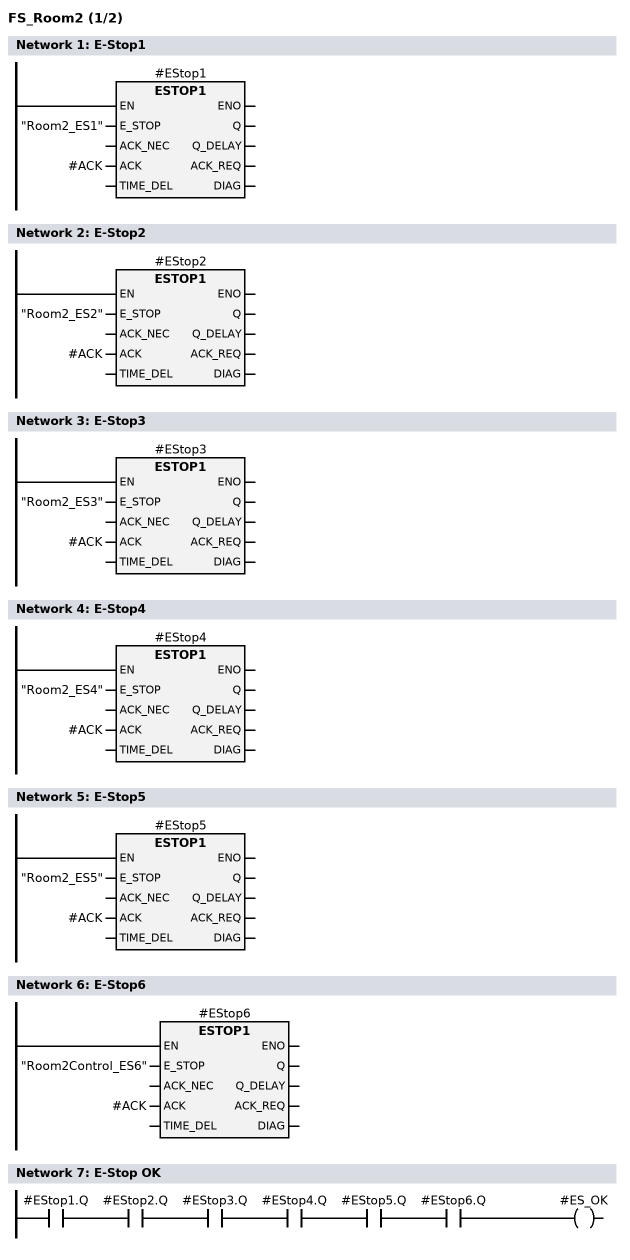
   RUNG wire#powerrail
      #EStop1.ESTOP1(E_STOP := "Room2_ES1", ACK_NEC :=, ACK := #ACK, TIME_DEL :=, Q =>, Q_DELAY =>, ACK_REQ =>, DIAG =>)
   END_RUNG
   // the same network as SCL:
   #EStop1(E_STOP := "Room2_ES1", ACK := #ACK);   // ESTOP1
END_REGION

REGION Network 2: E-Stop2
   RUNG wire#powerrail
      #EStop2.ESTOP1(E_STOP := "Room2_ES2", ACK_NEC :=, ACK := #ACK, TIME_DEL :=, Q =>, Q_DELAY =>, ACK_REQ =>, DIAG =>)
   END_RUNG
   // the same network as SCL:
   #EStop2(E_STOP := "Room2_ES2", ACK := #ACK);   // ESTOP1
END_REGION

REGION Network 3: E-Stop3
   RUNG wire#powerrail
      #EStop3.ESTOP1(E_STOP := "Room2_ES3", ACK_NEC :=, ACK := #ACK, TIME_DEL :=, Q =>, Q_DELAY =>, ACK_REQ =>, DIAG =>)
   END_RUNG
   // the same network as SCL:
   #EStop3(E_STOP := "Room2_ES3", ACK := #ACK);   // ESTOP1
END_REGION

REGION Network 4: E-Stop4
   RUNG wire#powerrail
      #EStop4.ESTOP1(E_STOP := "Room2_ES4", ACK_NEC :=, ACK := #ACK, TIME_DEL :=, Q =>, Q_DELAY =>, ACK_REQ =>, DIAG =>)
   END_RUNG
   // the same network as SCL:
   #EStop4(E_STOP := "Room2_ES4", ACK := #ACK);   // ESTOP1
END_REGION

REGION Network 5: E-Stop5
   RUNG wire#powerrail
      #EStop5.ESTOP1(E_STOP := "Room2_ES5", ACK_NEC :=, ACK := #ACK, TIME_DEL :=, Q =>, Q_DELAY =>, ACK_REQ =>, DIAG =>)
   END_RUNG
   // the same network as SCL:
   #EStop5(E_STOP := "Room2_ES5", ACK := #ACK);   // ESTOP1
END_REGION

REGION Network 6: E-Stop6
   RUNG wire#powerrail
      #EStop6.ESTOP1(E_STOP := "Room2Control_ES6", ACK_NEC :=, ACK := #ACK, TIME_DEL :=, Q =>, Q_DELAY =>, ACK_REQ =>, DIAG =>)
   END_RUNG
   // the same network as SCL:
   #EStop6(E_STOP := "Room2Control_ES6", ACK := #ACK);   // ESTOP1
END_REGION

REGION Network 7: E-Stop OK
   RUNG wire#powerrail
      Contact( #EStop1.Q )
      Contact( #EStop2.Q )
      Contact( #EStop3.Q )
      Contact( #EStop4.Q )
      Contact( #EStop5.Q )
      Contact( #EStop6.Q )
      Coil( #ES_OK )
   END_RUNG
   // the same network as SCL:
   #ES_OK := #EStop1.Q AND #EStop2.Q AND #EStop3.Q AND #EStop4.Q AND #EStop5.Q AND #EStop6.Q;
END_REGION

REGION Network 8: door
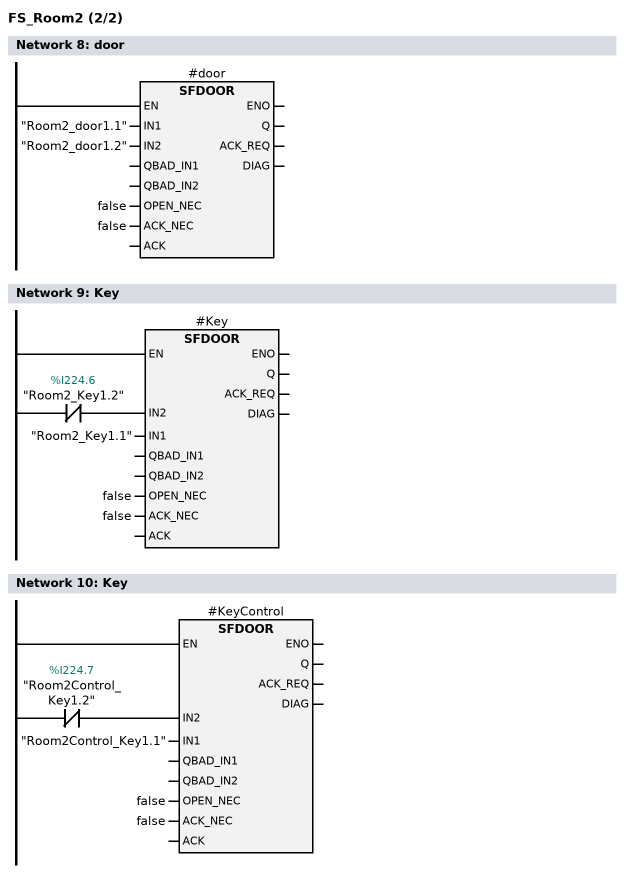
   RUNG wire#powerrail
      #door.SFDOOR(IN1 := "Room2_door1.1", IN2 := "Room2_door1.2", QBAD_IN1 :=, QBAD_IN2 :=, OPEN_NEC := false, ACK_NEC := false, ACK :=, Q =>, ACK_REQ =>, DIAG =>)
   END_RUNG
   // the same network as SCL:
   #door(IN1 := "Room2_door1.1", IN2 := "Room2_door1.2", OPEN_NEC := false, ACK_NEC := false);   // SFDOOR
END_REGION

REGION Network 9: Key
   RUNG wire#powerrail
      #Key.SFDOOR(IN2 := wire#w1, IN1 := "Room2_Key1.1", QBAD_IN1 :=, QBAD_IN2 :=, OPEN_NEC := false, ACK_NEC := false, ACK :=, Q =>, ACK_REQ =>, DIAG =>)
   END_RUNG
   RUNG wire#powerrail
      I_Contact( "Room2_Key1.2" )
   END_RUNG wire#w1
   // the same network as SCL:
   #Key(IN2 := NOT "Room2_Key1.2", IN1 := "Room2_Key1.1", OPEN_NEC := false, ACK_NEC := false);   // SFDOOR
END_REGION

REGION Network 10: Key
   RUNG wire#powerrail
      #KeyControl.SFDOOR(IN2 := wire#w1, IN1 := "Room2Control_Key1.1", QBAD_IN1 :=, QBAD_IN2 :=, OPEN_NEC := false, ACK_NEC := false, ACK :=, Q =>, ACK_REQ =>, DIAG =>)
   END_RUNG
   RUNG wire#powerrail
      I_Contact( "Room2Control_Key1.2" )
   END_RUNG wire#w1
   // the same network as SCL:
   #KeyControl(IN2 := NOT "Room2Control_Key1.2",   // SFDOOR
               IN1 := "Room2Control_Key1.1",
               OPEN_NEC := false,
               ACK_NEC := false);
END_REGION
END_FUNCTION_BLOCK

FUNCTION_BLOCK "FS_VerticalBeam"   // FB5, F_LAD
{ S7_Optimized_Access := 'TRUE' }
VERSION : 0.1
// stored: AutoNumber false, IsIECCheckEnabled false, UDAEnableTagReadback false
   VAR_INPUT
      ACK : Bool;
   END_VAR
   VAR_OUTPUT
      ES_OK : Bool;
   END_VAR
   VAR
      EStop1 { S7_SetPoint := 'True'} : ESTOP1;
      EStop2 { S7_SetPoint := 'True'} : ESTOP1;
      EStop3 { S7_SetPoint := 'True'} : ESTOP1;
      EStop4 { S7_SetPoint := 'True'} : ESTOP1;
      door1 : SFDOOR;
      door2 : SFDOOR;
      Key : SFDOOR;
      KeyControl : SFDOOR;
   END_VAR
BEGIN

REGION Network 1: E-Stop1
